KUKA KRL program: MyProgram_197().src

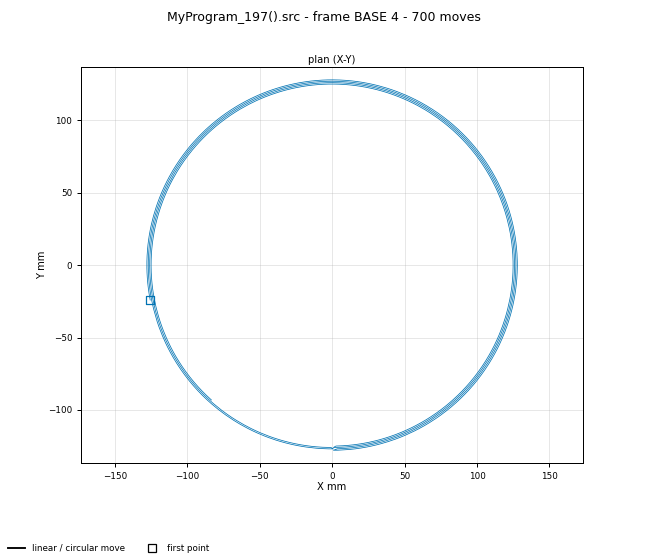
[picture p0: tool path of MyProgram_197().src in frame BASE 4, 700 of 700 moves have a stored position in this frame; points joined in program order, loops and branches not executed]
&ACCESS RVP
&REL 1
&PARAM TEMPLATE = C:\KRC\Roboter\Template\vorgabe
&PARAM EDITMASK = *
DEF MyProgram_197()
; ---- Setting reference (Base) ----
$BASE = BASE_DATA[4]

; --------------------------
; ---- Setting tool (TCP) ----
$TOOL = TOOL_DATA[3]
; --------------------------

$VEL.CP = VEL_APROX_PRINT
Startdeposition()
$VEL.CP = VEL_PRINT
LIN {X -125.5211,Y -24.1311,Z 142,A -173.0115,B 24.959,C -1.4779,E1 24.8425,E2 259.4302} C_DIS
LIN {X -126.2211,Y -20.1609,Z 142,A -174.9442,B 24.959,C -1.4779,E1 24.8416,E2 261.3743} C_DIS
LIN {X -126.7719,Y -16.3344,Z 142,A -176.6253,B 24.9586,C -1.4859,E1 24.841,E2 263.0464} C_DIS
LIN {X -127.2142,Y -12.4288,Z 142,A -178.3522,B 24.9582,C -1.4932,E1 24.8404,E2 264.7662} C_DIS
LIN {X -127.5104,Y -8.8962,Z 142,A 179.9691,B 24.9582,C -1.4943,E1 24.8401,E2 266.4524} C_DIS
LIN {X -127.7137,Y -5.2116,Z 142,A 178.4133,B 24.9576,C -1.5042,E1 24.8399,E2 267.994} C_DIS
LIN {X -127.8085,Y -1.741,Z 142,A 176.7456,B 24.9576,C -1.5042,E1 24.8398,E2 269.6717} C_DIS
LIN {X -127.7955,Y 2.5271,Z 142,A 174.7944,B 24.9573,C -1.5088,E1 24.8398,E2 271.6238} C_DIS
LIN {X -127.6549,Y 6.4899,Z 142,A 173.0449,B 24.9569,C -1.516,E1 24.8401,E2 273.3668} C_DIS
LIN {X -127.3797,Y 10.5984,Z 142,A 171.2555,B 24.9565,C -1.5246,E1 24.8404,E2 275.1463} C_DIS
LIN {X -127.0589,Y 13.9273,Z 142,A 169.9088,B 24.9558,C -1.5365,E1 24.8408,E2 276.4728} C_DIS
LIN {X -126.6556,Y 17.2223,Z 142,A 168.2535,B 24.9559,C -1.5337,E1 24.8414,E2 278.1446} C_DIS
LIN {X -126.1339,Y 20.693,Z 142,A 166.6904,B 24.9556,C -1.5393,E1 24.8421,E2 279.7035} C_DIS
LIN {X -125.5309,Y 24.0797,Z 142,A 165.0614,B 24.9556,C -1.5404,E1 24.8429,E2 281.3395} C_DIS
LIN {X -124.7397,Y 27.8958,Z 142,A 163.305,B 24.9552,C -1.5457,E1 24.8439,E2 283.0938} C_DIS
LIN {X -123.2875,Y 33.7418,Z 142,A 159.7071,B 24.9571,C -1.514,E1 24.8466,E2 286.7881} C_DIS
LIN {X -121.4906,Y 39.7278,Z 142,A 157.6719,B 24.9546,C -1.5574,E1 24.8482,E2 288.7316} C_DIS
LIN {X -120.38,Y 42.9722,Z 142,A 156.2415,B 24.954,C -1.5671,E1 24.8495,E2 290.147} C_DIS
LIN {X -119.1546,Y 46.2598,Z 142,A 154.6827,B 24.9537,C -1.5727,E1 24.8511,E2 291.7012} C_DIS
LIN {X -117.5968,Y 50.0924,Z 142,A 152.5641,B 24.954,C -1.5665,E1 24.8534,E2 293.8465} C_DIS
LIN {X -115.5684,Y 54.6078,Z 142,A 150.536,B 24.9531,C -1.582,E1 24.8557,E2 295.8487} C_DIS
LIN {X -113.9888,Y 57.8302,Z 142,A 148.9277,B 24.9528,C -1.5869,E1 24.8577,E2 297.454} C_DIS
LIN {X -112.4203,Y 60.8282,Z 142,A 147.428,B 24.9525,C -1.5921,E1 24.8597,E2 298.9491} C_DIS
LIN {X -109.9142,Y 65.2469,Z 142,A 145.041,B 24.9525,C -1.5938,E1 24.863,E2 301.3445} C_DIS
LIN {X -107.564,Y 69.0526,Z 142,A 143.0449,B 24.952,C -1.6001,E1 24.866,E2 303.3359} C_DIS
LIN {X -105.1568,Y 72.6668,Z 142,A 141.0404,B 24.9519,C -1.6029,E1 24.8691,E2 305.3436} C_DIS
LIN {X -102.5814,Y 76.2581,Z 142,A 139.0821,B 24.9515,C -1.6095,E1 24.8723,E2 307.2957} C_DIS
LIN {X -99.8212,Y 79.8378,Z 142,A 137.0452,B 24.9512,C -1.6144,E1 24.8758,E2 309.3304} C_DIS
LIN {X -97.6988,Y 82.4216,Z 142,A 135.4913,B 24.9511,C -1.6159,E1 24.8786,E2 310.888} C_DIS
LIN {X -95.3727,Y 85.1019,Z 142,A 133.294,B 24.9525,C -1.5923,E1 24.8829,E2 313.1512} C_DIS
LIN {X -91.7521,Y 88.9933,Z 142,A 130.8212,B 24.9524,C -1.5942,E1 24.8877,E2 315.6302} C_DIS
LIN {X -87.6911,Y 92.9974,Z 142,A 129.1164,B 24.9496,C -1.6394,E1 24.8909,E2 317.2346} C_DIS
LIN {X -85.5377,Y 94.9821,Z 142,A 127.2535,B 24.951,C -1.6171,E1 24.8949,E2 319.1579} C_DIS
LIN {X -82.4213,Y 97.6989,Z 142,A 125.4338,B 24.9507,C -1.6228,E1 24.8987,E2 320.971} C_DIS
LIN {X -79.4084,Y 100.1629,Z 142,A 124.047,B 24.9494,C -1.6432,E1 24.9017,E2 322.3146} C_DIS
LIN {X -76.1096,Y 102.6921,Z 142,A 122.2381,B 24.949,C -1.6497,E1 24.9057,E2 324.1145} C_DIS
LIN {X -73.0168,Y 104.9132,Z 142,A 120.494,B 24.9489,C -1.6515,E1 24.9097,E2 325.8603} C_DIS
LIN {X -69.7238,Y 107.1301,Z 142,A 118.719,B 24.9487,C -1.6552,E1 24.9138,E2 327.6323} C_DIS
LIN {X -66.2948,Y 109.2853,Z 142,A 117.1421,B 24.9477,C -1.6698,E1 24.9175,E2 329.1794} C_DIS
LIN {X -63.6066,Y 110.8718,Z 142,A 115.4076,B 24.9486,C -1.6567,E1 24.9217,E2 330.9504} C_DIS
LIN {X -59.9113,Y 112.9101,Z 142,A 113.5668,B 24.9482,C -1.6624,E1 24.9262,E2 332.7828} C_DIS
LIN {X -56.6117,Y 114.5988,Z 142,A 111.9713,B 24.9478,C -1.6682,E1 24.9302,E2 334.3687} C_DIS
LIN {X -53.8031,Y 115.944,Z 142,A 110.6023,B 24.9476,C -1.6717,E1 24.9336,E2 335.7329} C_DIS
LIN {X -50.9119,Y 117.2424,Z 142,A 109.1599,B 24.9476,C -1.6728,E1 24.9373,E2 337.1761} C_DIS
LIN {X -47.8666,Y 118.5182,Z 142,A 107.9143,B 24.9467,C -1.6861,E1 24.9405,E2 338.393} C_DIS
LIN {X -43.9077,Y 120.0427,Z 142,A 105.6564,B 24.9476,C -1.6717,E1 24.9465,E2 340.6897} C_DIS
LIN {X -40.618,Y 121.1942,Z 142,A 104.4038,B 24.9466,C -1.6884,E1 24.9497,E2 341.9052} C_DIS
LIN {X -36.1428,Y 122.6033,Z 142,A 102.1604,B 24.9468,C -1.6841,E1 24.9557,E2 344.1626} C_DIS
LIN {X -33.0254,Y 123.4793,Z 142,A 100.6082,B 24.9471,C -1.6809,E1 24.9599,E2 345.725} C_DIS
LIN {X -29.441,Y 124.3838,Z 142,A 98.9805,B 24.9469,C -1.6839,E1 24.9643,E2 347.3478} C_DIS
LIN {X -25.4757,Y 125.255,Z 142,A 97.1695,B 24.9467,C -1.6859,E1 24.9692,E2 349.1562} C_DIS
LIN {X -22.4451,Y 125.8335,Z 142,A 95.7361,B 24.9468,C -1.6846,E1 24.9732,E2 350.5942} C_DIS
LIN {X -18.4345,Y 126.4838,Z 142,A 93.8652,B 24.9468,C -1.6835,E1 24.9783,E2 352.4694} C_DIS
LIN {X -14.5682,Y 126.9881,Z 142,A 92.0699,B 24.947,C -1.6822,E1 24.9833,E2 354.2689} C_DIS
LIN {X -10.682,Y 127.3726,Z 142,A 90.406,B 24.9467,C -1.6873,E1 24.9879,E2 355.9217} C_DIS
LIN {X -6.5608,Y 127.6514,Z 142,A 88.2139,B 24.9476,C -1.6716,E1 24.9941,E2 358.1517} C_DIS
LIN {X -3.06,Y 127.7841,Z 142,A 86.8826,B 24.9469,C -1.6835,E1 24.9978,E2 359.4548} C_DIS
LIN {X 0.8422,Y 127.8171,Z 142,A 84.6902,B 24.9482,C -1.6625,E1 25.0041,E2 361.6969} C_DIS
LIN {X 5.3004,Y 127.7102,Z 142,A 83.2635,B 24.9465,C -1.6903,E1 25.0079,E2 363.0573} C_DIS
LIN {X 9.2581,Y 127.484,Z 142,A 81.399,B 24.9467,C -1.686,E1 25.0131,E2 364.9312} C_DIS
LIN {X 13.5575,Y 127.0987,Z 142,A 79.5233,B 24.9466,C -1.6887,E1 25.0183,E2 366.7994} C_DIS
LIN {X 17.3749,Y 126.6352,Z 142,A 77.688,B 24.9469,C -1.6828,E1 25.0234,E2 368.6472} C_DIS
LIN {X 21.1329,Y 126.0605,Z 142,A 76.0592,B 24.9467,C -1.686,E1 25.0278,E2 370.2669} C_DIS
LIN {X 25.2748,Y 125.2959,Z 142,A 74.3916,B 24.9461,C -1.696,E1 25.0323,E2 371.9087} C_DIS
LIN {X 28.2787,Y 124.6522,Z 142,A 72.7974,B 24.9468,C -1.6846,E1 25.0368,E2 373.5279} C_DIS
LIN {X 32.0392,Y 123.7404,Z 142,A 71.1216,B 24.9468,C -1.6864,E1 25.0413,E2 375.1969} C_DIS
LIN {X 35.599,Y 122.7625,Z 142,A 69.4783,B 24.9468,C -1.6859,E1 25.0457,E2 376.8388} C_DIS
LIN {X 38.0718,Y 122.0198,Z 142,A 68.3592,B 24.9467,C -1.6868,E1 25.0487,E2 377.9535} C_DIS
LIN {X 41.211,Y 120.9956,Z 142,A 66.7028,B 24.9473,C -1.6768,E1 25.0531,E2 379.6305} C_DIS
LIN {X 44.792,Y 119.7141,Z 142,A 65.2062,B 24.9468,C -1.6856,E1 25.057,E2 381.1031} C_DIS
LIN {X 50.6604,Y 117.3512,Z 142,A 62.3209,B 24.9471,C -1.6801,E1 25.0645,E2 383.9949} C_DIS
LIN {X 53.5915,Y 116.0419,Z 142,A 60.9427,B 24.9471,C -1.6815,E1 25.0679,E2 385.3665} C_DIS
LIN {X 57.6244,Y 114.0936,Z 142,A 58.835,B 24.9475,C -1.6739,E1 25.0733,E2 387.4864} C_DIS
LIN {X 60.9743,Y 112.3408,Z 142,A 57.0504,B 24.9479,C -1.667,E1 25.0777,E2 389.2823} C_DIS
LIN {X 65.0173,Y 110.0504,Z 142,A 54.8897,B 24.9484,C -1.66,E1 25.0829,E2 391.4529} C_DIS
LIN {X 69.2753,Y 107.4213,Z 142,A 52.7962,B 24.9481,C -1.664,E1 25.0878,E2 393.5303} C_DIS
LIN {X 73.0165,Y 104.9135,Z 142,A 50.8001,B 24.9483,C -1.6618,E1 25.0924,E2 395.5248} C_DIS
LIN {X 76.4508,Y 102.438,Z 142,A 48.8884,B 24.9485,C -1.6577,E1 25.0968,E2 397.4395} C_DIS
LIN {X 79.9444,Y 99.7361,Z 142,A 46.8456,B 24.9489,C -1.6507,E1 25.1013,E2 399.4911} C_DIS
LIN {X 83.3953,Y 96.8683,Z 142,A 44.9121,B 24.9489,C -1.6507,E1 25.1054,E2 401.417} C_DIS
LIN {X 86.719,Y 93.9049,Z 142,A 42.9267,B 24.9492,C -1.6472,E1 25.1095,E2 403.4029} C_DIS
LIN {X 89.7869,Y 90.9764,Z 142,A 40.9805,B 24.9496,C -1.6408,E1 25.1134,E2 405.356} C_DIS
LIN {X 92.8123,Y 87.8873,Z 142,A 39.056,B 24.9498,C -1.6372,E1 25.1171,E2 407.2808} C_DIS
LIN {X 95.8563,Y 84.5567,Z 142,A 37.1194,B 24.9498,C -1.6369,E1 25.1207,E2 409.2094} C_DIS
LIN {X 98.6264,Y 81.309,Z 142,A 35.3653,B 24.9496,C -1.6406,E1 25.1238,E2 410.9469} C_DIS
LIN {X 100.8028,Y 78.595,Z 142,A 33.5657,B 24.9506,C -1.6243,E1 25.127,E2 412.7764} C_DIS
LIN {X 103.5568,Y 74.9283,Z 142,A 31.6066,B 24.9506,C -1.6241,E1 25.1303,E2 414.7265} C_DIS
LIN {X 106.0451,Y 71.3639,Z 142,A 29.6102,B 24.951,C -1.6166,E1 25.1334,E2 416.7309} C_DIS
LIN {X 108.3748,Y 67.7734,Z 142,A 27.867,B 24.9508,C -1.6206,E1 25.136,E2 418.456} C_DIS
LIN {X 110.4975,Y 64.2543,Z 142,A 25.882,B 24.9515,C -1.6081,E1 25.1389,E2 420.46} C_DIS
LIN {X 112.6207,Y 60.4551,Z 142,A 23.9087,B 24.9519,C -1.6015,E1 25.1415,E2 422.4386} C_DIS
LIN {X 114.4624,Y 56.8881,Z 142,A 22.0946,B 24.9523,C -1.5957,E1 25.1438,E2 424.2568} C_DIS
LIN {X 116.4788,Y 52.6375,Z 142,A 20.1062,B 24.9523,C -1.5958,E1 25.1461,E2 426.2341} C_DIS
LIN {X 118.1644,Y 48.7368,Z 142,A 17.8754,B 24.9536,C -1.5732,E1 25.1486,E2 428.506} C_DIS
LIN {X 119.5011,Y 45.3606,Z 142,A 16.5973,B 24.9528,C -1.5865,E1 25.1498,E2 429.7456} C_DIS
LIN {X 120.711,Y 42.032,Z 142,A 15.1443,B 24.9528,C -1.5888,E1 25.1512,E2 431.1852} C_DIS
LIN {X 122.3547,Y 36.9776,Z 142,A 12.5736,B 24.9537,C -1.5716,E1 25.1534,E2 433.7818} C_DIS
LIN {X 123.4571,Y 33.1089,Z 142,A 10.9486,B 24.9535,C -1.5753,E1 25.1546,E2 435.3887} C_DIS
LIN {X 124.253,Y 29.9836,Z 142,A 9.4672,B 24.9539,C -1.5689,E1 25.1556,E2 436.8767} C_DIS
LIN {X 125.0962,Y 26.2549,Z 142,A 7.6746,B 24.9544,C -1.5593,E1 25.1567,E2 438.6815} C_DIS
LIN {X 125.7954,Y 22.6581,Z 142,A 6.1398,B 24.9544,C -1.5597,E1 25.1574,E2 440.2063} C_DIS
LIN {X 126.3274,Y 19.4745,Z 142,A 4.6884,B 24.9547,C -1.5548,E1 25.1581,E2 441.6608} C_DIS
LIN {X 126.8738,Y 15.526,Z 142,A 2.8912,B 24.9551,C -1.5485,E1 25.1587,E2 443.4623} C_DIS
LIN {X 127.2651,Y 11.8982,Z 142,A 1.1815,B 24.9556,C -1.5392,E1 25.1592,E2 445.1836} C_DIS
LIN {X 127.5819,Y 7.7944,Z 142,A -0.2836,B 24.9548,C -1.5533,E1 25.1595,E2 446.607} C_DIS
LIN {X 127.7943,Y 2.5998,Z 142,A -2.9024,B 24.9561,C -1.5303,E1 25.1598,E2 449.2642} C_DIS
LIN {X 127.8184,Y -0.7537,Z 142,A -4.9005,B 24.9579,C -1.4994,E1 25.1598,E2 451.3233} C_DIS
LIN {X 127.7126,Y -5.24,Z 142,A -6.8008,B 24.9579,C -1.4986,E1 25.1595,E2 453.2143} C_DIS
LIN {X 127.4849,Y -9.2456,Z 142,A -8.1262,B 24.9569,C -1.5175,E1 25.1593,E2 454.4872} C_DIS
LIN {X 127.1509,Y -13.0722,Z 142,A -9.9525,B 24.9575,C -1.5063,E1 25.1588,E2 456.3291} C_DIS
LIN {X 126.6224,Y -17.4646,Z 142,A -11.7547,B 24.9573,C -1.5093,E1 25.1582,E2 458.1136} C_DIS
LIN {X 126.2121,Y -20.2188,Z 142,A -13.1455,B 24.958,C -1.4976,E1 25.1576,E2 459.5237} C_DIS
LIN {X 125.5286,Y -24.0917,Z 142,A -14.7731,B 24.958,C -1.499,E1 25.1568,E2 461.1385} C_DIS
LIN {X 124.7218,Y -27.9739,Z 142,A -16.5708,B 24.9583,C -1.4921,E1 25.1557,E2 462.9419} C_DIS
LIN {X 123.9309,Y -31.2888,Z 142,A -18.0523,B 24.9584,C -1.4896,E1 25.1547,E2 464.4208} C_DIS
LIN {X 123.1029,Y -34.402,Z 142,A -19.499,B 24.9587,C -1.4848,E1 25.1537,E2 465.8705} C_DIS
LIN {X 121.7562,Y -38.9003,Z 142,A -21.5091,B 24.9587,C -1.483,E1 25.152,E2 467.8734} C_DIS
LIN {X 120.8724,Y -41.5664,Z 142,A -22.6636,B 24.9587,C -1.4845,E1 25.151,E2 469.0179} C_DIS
LIN {X 119.2673,Y -45.9699,Z 142,A -25.5916,B 24.9615,C -1.4344,E1 25.148,E2 472.0476} C_DIS
LIN {X 117.3926,Y -50.5645,Z 142,A -27.6944,B 24.9615,C -1.4338,E1 25.1457,E2 474.1403} C_DIS
LIN {X 115.5438,Y -54.6593,Z 142,A -29.2089,B 24.9604,C -1.4538,E1 25.144,E2 475.5996} C_DIS
LIN {X 113.976,Y -57.8555,Z 142,A -30.7502,B 24.9605,C -1.4518,E1 25.1421,E2 477.1373} C_DIS
LIN {X 112.2793,Y -61.0871,Z 142,A -32.4087,B 24.9608,C -1.4456,E1 25.1399,E2 478.8016} C_DIS
LIN {X 110.2445,Y -64.6869,Z 142,A -34.2573,B 24.9611,C -1.4404,E1 25.1373,E2 480.6529} C_DIS
LIN {X 107.9456,Y -68.4548,Z 142,A -36.8227,B 24.9631,C -1.404,E1 25.1334,E2 483.2912} C_DIS
LIN {X 105.1875,Y -72.6221,Z 142,A -38.4797,B 24.9618,C -1.428,E1 25.1309,E2 484.8835} C_DIS
LIN {X 102.7157,Y -76.0778,Z 142,A -40.3737,B 24.9621,C -1.4232,E1 25.1278,E2 486.7796} C_DIS
LIN {X 99.8994,Y -79.7395,Z 142,A -42.7564,B 24.9632,C -1.4013,E1 25.1236,E2 489.2029} C_DIS
LIN {X 97.5112,Y -82.6429,Z 142,A -44.2335,B 24.9629,C -1.4076,E1 25.121,E2 490.6583} C_DIS
LIN {X 94.3141,Y -86.2739,Z 142,A -46.2515,B 24.9628,C -1.4098,E1 25.1172,E2 492.6621} C_DIS
LIN {X 91.4762,Y -89.2773,Z 142,A -48.1018,B 24.963,C -1.4052,E1 25.1136,E2 494.5152} C_DIS
LIN {X 88.7083,Y -92.028,Z 142,A -49.9167,B 24.9634,C -1.3975,E1 25.11,E2 496.3409} C_DIS
LIN {X 85.397,Y -95.1085,Z 142,A -51.8738,B 24.9634,C -1.3963,E1 25.106,E2 498.2929} C_DIS
LIN {X 82.0889,Y -97.9779,Z 142,A -53.7796,B 24.9636,C -1.3947,E1 25.1019,E2 500.1949} C_DIS
LIN {X 79.0225,Y -100.4674,Z 142,A -55.7429,B 24.9643,C -1.3808,E1 25.0976,E2 502.1838} C_DIS
LIN {X 74.8412,Y -103.6199,Z 142,A -57.9197,B 24.9641,C -1.3845,E1 25.0927,E2 504.3439} C_DIS
LIN {X 71.4919,Y -105.9584,Z 142,A -59.5222,B 24.9637,C -1.3926,E1 25.0891,E2 505.9219} C_DIS
LIN {X 67.4024,Y -108.6056,Z 142,A -61.9092,B 24.9644,C -1.3778,E1 25.0834,E2 508.3361} C_DIS
LIN {X 63.7647,Y -110.7809,Z 142,A -63.7764,B 24.9645,C -1.3759,E1 25.0789,E2 510.2021} C_DIS
LIN {X 60.2915,Y -112.7086,Z 142,A -65.5892,B 24.9648,C -1.3711,E1 25.0745,E2 512.021} C_DIS
LIN {X 56.7055,Y -114.5525,Z 142,A -67.2969,B 24.9647,C -1.3732,E1 25.0702,E2 513.7192} C_DIS
LIN {X 53.6446,Y -116.0173,Z 142,A -68.7914,B 24.9647,C -1.3721,E1 25.0665,E2 515.2124} C_DIS
LIN {X 50.9167,Y -117.2404,Z 142,A -70.604,B 24.9661,C -1.3459,E1 25.0617,E2 517.0824} C_DIS
LIN {X 47.1355,Y -118.8129,Z 142,A -72.1159,B 24.9654,C -1.3597,E1 25.0579,E2 518.5583} C_DIS
LIN {X 43.615,Y -120.1482,Z 142,A -73.5663,B 24.9649,C -1.3695,E1 25.0541,E2 519.9824} C_DIS
LIN {X 38.4751,Y -121.892,Z 142,A -76.206,B 24.9656,C -1.3559,E1 25.0471,E2 522.6493} C_DIS
LIN {X 33.9823,Y -123.2202,Z 142,A -78.2965,B 24.9656,C -1.354,E1 25.0415,E2 524.7407} C_DIS
LIN {X 30.1126,Y -124.2219,Z 142,A -79.9655,B 24.9654,C -1.3584,E1 25.037,E2 526.3969} C_DIS
LIN {X 27.1122,Y -124.9111,Z 142,A -81.3455,B 24.9655,C -1.3571,E1 25.0332,E2 527.7781} C_DIS
LIN {X 23.7699,Y -125.5902,Z 142,A -82.9365,B 24.9657,C -1.3526,E1 25.0288,E2 529.3778} C_DIS
LIN {X 19.7669,Y -126.2821,Z 142,A -84.7048,B 24.9657,C -1.3539,E1 25.024,E2 531.1413} C_DIS
LIN {X 16.1602,Y -126.7948,Z 142,A -86.226,B 24.9654,C -1.3584,E1 25.0198,E2 532.6505} C_DIS
LIN {X 11.938,Y -127.2613,Z 142,A -88.2251,B 24.9657,C -1.3525,E1 25.0142,E2 534.6622} C_DIS
LIN {X 4.0063,Y -127.7578,Z 142,A -91.6254,B 24.9654,C -1.3591,E1 25.0048,E2 538.0457} C_DIS
LIN {X 0.9092,Y -127.7876,Z 142,A -93.0254,B 24.9654,C -1.3586,E1 25.0009,E2 539.4466} C_DIS
Enddeposition()
LIN {X 0.9092,Y -127.7876,Z 142,A -93.0254,B 24.9654,C -1.3586,E1 25.0009,E2 539.4466} C_DIS
Startdeposition()
$VEL.CP = VEL_PRINT
LIN {X 3.5824,Y -126.8,Z 142,A -91.1897,B 24.4984,C -1.3089,E1 24.537,E2 537.666} C_DIS
LIN {X 9.8682,Y -126.4677,Z 142,A -88.1818,B 24.498,C -1.3182,E1 24.5455,E2 534.6369} C_DIS
LIN {X 12.9375,Y -126.1906,Z 142,A -86.8649,B 24.4981,C -1.3153,E1 24.5491,E2 533.328} C_DIS
LIN {X 16.3259,Y -125.7956,Z 142,A -85.3641,B 24.4981,C -1.3143,E1 24.5533,E2 531.8307} C_DIS
LIN {X 20.2934,Y -125.218,Z 142,A -83.4855,B 24.4979,C -1.3189,E1 24.5585,E2 529.9428} C_DIS
LIN {X 23.9684,Y -124.5655,Z 142,A -81.8724,B 24.498,C -1.3167,E1 24.5629,E2 528.3369} C_DIS
LIN {X 28.0075,Y -123.72,Z 142,A -80.0259,B 24.498,C -1.3176,E1 24.5679,E2 526.4907} C_DIS
LIN {X 31.241,Y -122.9431,Z 142,A -78.5522,B 24.498,C -1.3176,E1 24.5719,E2 525.0191} C_DIS
LIN {X 34.1426,Y -122.169,Z 142,A -76.8134,B 24.4969,C -1.3383,E1 24.5767,E2 523.2335} C_DIS
LIN {X 37.5906,Y -121.1535,Z 142,A -75.6621,B 24.4981,C -1.3165,E1 24.5797,E2 522.1368} C_DIS
LIN {X 44.5342,Y -118.7757,Z 142,A -72.2474,B 24.4976,C -1.3257,E1 24.5887,E2 518.7069} C_DIS
LIN {X 47.4707,Y -117.6329,Z 142,A -70.2624,B 24.496,C -1.3562,E1 24.594,E2 516.6532} C_DIS
LIN {X 51.6656,Y -115.8517,Z 142,A -68.7876,B 24.4974,C -1.3297,E1 24.5976,E2 515.2457} C_DIS
LIN {X 54.574,Y -114.5104,Z 142,A -67.3594,B 24.4974,C -1.3311,E1 24.6012,E2 513.818} C_DIS
LIN {X 57.4301,Y -113.105,Z 142,A -65.9894,B 24.4974,C -1.3301,E1 24.6046,E2 512.4541} C_DIS
LIN {X 60.4982,Y -111.4965,Z 142,A -64.2484,B 24.4968,C -1.3417,E1 24.609,E2 510.6903} C_DIS
LIN {X 64.3963,Y -109.2912,Z 142,A -62.2671,B 24.4967,C -1.3433,E1 24.6137,E2 508.7112} C_DIS
LIN {X 68.0897,Y -107.0296,Z 142,A -60.3105,B 24.4965,C -1.3471,E1 24.6184,E2 506.7519} C_DIS
LIN {X 75.4232,Y -101.9947,Z 142,A -55.6797,B 24.4944,C -1.3869,E1 24.6291,E2 502.0419} C_DIS
LIN {X 79.5373,Y -98.8192,Z 142,A -53.9974,B 24.4959,C -1.3578,E1 24.6326,E2 500.4359} C_DIS
LIN {X 82.7212,Y -96.1698,Z 142,A -52.1009,B 24.4956,C -1.3634,E1 24.6367,E2 498.5335} C_DIS
LIN {X 86.0309,Y -93.221,Z 142,A -49.7721,B 24.4945,C -1.385,E1 24.6416,E2 496.1624} C_DIS
LIN {X 88.7862,Y -90.6004,Z 142,A -48.3236,B 24.495,C -1.3753,E1 24.6444,E2 494.7434} C_DIS
LIN {X 92.0815,Y -87.2496,Z 142,A -46.2633,B 24.495,C -1.3774,E1 24.6484,E2 492.687} C_DIS
LIN {X 94.7896,Y -84.3,Z 142,A -44.0129,B 24.4934,C -1.405,E1 24.6527,E2 490.3807} C_DIS
LIN {X 97.7119,Y -80.8938,Z 142,A -41.8235,B 24.4927,C -1.4189,E1 24.6566,E2 488.1683} C_DIS
LIN {X 101.0638,Y -76.6654,Z 142,A -40.0221,B 24.4941,C -1.3925,E1 24.6596,E2 486.439} C_DIS
LIN {X 103.4919,Y -73.3547,Z 142,A -37.2766,B 24.4913,C -1.4442,E1 24.6642,E2 483.5831} C_DIS
LIN {X 107.259,Y -67.7268,Z 142,A -35.1816,B 24.4936,C -1.4025,E1 24.6672,E2 481.5988} C_DIS
LIN {X 109.5043,Y -64.0336,Z 142,A -33.2445,B 24.4933,C -1.4075,E1 24.6699,E2 479.66} C_DIS
LIN {X 111.5832,Y -60.3384,Z 142,A -31.2807,B 24.4929,C -1.4157,E1 24.6726,E2 477.6869} C_DIS
LIN {X 113.6319,Y -56.3809,Z 142,A -29.4244,B 24.4929,C -1.4137,E1 24.6749,E2 475.8456} C_DIS
LIN {X 116.1307,Y -51.0383,Z 142,A -26.3133,B 24.4912,C -1.4452,E1 24.6786,E2 472.6762} C_DIS
LIN {X 117.6366,Y -47.4613,Z 142,A -25.0374,B 24.4923,C -1.4257,E1 24.6799,E2 471.454} C_DIS
LIN {X 118.7903,Y -44.4951,Z 142,A -23.4782,B 24.4917,C -1.4366,E1 24.6814,E2 469.8778} C_DIS
LIN {X 120.3455,Y -40.0991,Z 142,A -21.558,B 24.4919,C -1.4336,E1 24.6832,E2 467.9757} C_DIS
LIN {X 121.8318,Y -35.3286,Z 142,A -19.1706,B 24.4911,C -1.4476,E1 24.6851,E2 465.5687} C_DIS
LIN {X 122.9124,Y -31.3619,Z 142,A -17.3901,B 24.491,C -1.4496,E1 24.6864,E2 463.7939} C_DIS
LIN {X 124.3904,Y -24.864,Z 142,A -14.3701,B 24.4904,C -1.4598,E1 24.6882,E2 460.7672} C_DIS
LIN {X 125.1064,Y -20.9624,Z 142,A -12.6537,B 24.4904,C -1.4618,E1 24.689,E2 459.0564} C_DIS
LIN {X 125.6936,Y -17.1039,Z 142,A -10.8449,B 24.4899,C -1.4699,E1 24.6897,E2 457.239} C_DIS
LIN {X 126.1566,Y -13.2533,Z 142,A -9.1161,B 24.4896,C -1.4745,E1 24.6903,E2 455.5096} C_DIS
LIN {X 126.5133,Y -9.2427,Z 142,A -7.3882,B 24.4896,C -1.4757,E1 24.6907,E2 453.7892} C_DIS
LIN {X 126.6899,Y -6.3824,Z 142,A -6.0741,B 24.4892,C -1.481,E1 24.6909,E2 452.4704} C_DIS
LIN {X 126.8523,Y -0.221,Z 142,A -3.1948,B 24.4884,C -1.4951,E1 24.691,E2 449.575} C_DIS
LIN {X 126.8205,Y 2.8402,Z 142,A -1.7619,B 24.488,C -1.5022,E1 24.691,E2 448.1337} C_DIS
LIN {X 126.6321,Y 7.4489,Z 142,A 0.1586,B 24.4881,C -1.5005,E1 24.6907,E2 446.2288} C_DIS
LIN {X 126.3715,Y 11.0191,Z 142,A 1.7934,B 24.4878,C -1.5067,E1 24.6903,E2 444.5891} C_DIS
LIN {X 125.9469,Y 15.1138,Z 142,A 3.6221,B 24.4875,C -1.5112,E1 24.6897,E2 442.7608} C_DIS
LIN {X 125.4053,Y 19.0953,Z 142,A 5.4185,B 24.4872,C -1.516,E1 24.689,E2 440.9636} C_DIS
LIN {X 124.8109,Y 22.6572,Z 142,A 7.0659,B 24.4869,C -1.5221,E1 24.6882,E2 439.3115} C_DIS
LIN {X 124.0247,Y 26.625,Z 142,A 8.838,B 24.4867,C -1.525,E1 24.6872,E2 437.5429} C_DIS
LIN {X 123.2119,Y 30.1668,Z 142,A 10.5459,B 24.4862,C -1.5336,E1 24.6861,E2 435.8245} C_DIS
LIN {X 122.0531,Y 34.557,Z 142,A 12.7063,B 24.4855,C -1.5457,E1 24.6845,E2 433.6479} C_DIS
LIN {X 119.6097,Y 42.2497,Z 142,A 16.1784,B 24.4854,C -1.5477,E1 24.6815,E2 430.1909} C_DIS
LIN {X 118.4151,Y 45.4869,Z 142,A 18.0658,B 24.4841,C -1.5694,E1 24.6796,E2 428.2622} C_DIS
LIN {X 117.0646,Y 48.8552,Z 142,A 19.2367,B 24.4852,C -1.5501,E1 24.6784,E2 427.1443} C_DIS
LIN {X 115.8591,Y 51.6491,Z 142,A 20.6227,B 24.4849,C -1.5547,E1 24.6768,E2 425.7549} C_DIS
LIN {X 114.5182,Y 54.5577,Z 142,A 21.8499,B 24.4854,C -1.5476,E1 24.6754,E2 424.5515} C_DIS
LIN {X 112.3862,Y 58.8243,Z 142,A 24.2286,B 24.4843,C -1.5651,E1 24.6724,E2 422.1436} C_DIS
LIN {X 110.4489,Y 62.3902,Z 142,A 26.6547,B 24.4822,C -1.6007,E1 24.669,E2 419.645} C_DIS
LIN {X 108.0931,Y 66.3875,Z 142,A 28.2209,B 24.4835,C -1.5791,E1 24.6668,E2 418.1389} C_DIS
LIN {X 105.8225,Y 69.9505,Z 142,A 30.1266,B 24.4832,C -1.584,E1 24.6639,E2 416.2312} C_DIS
LIN {X 103.0731,Y 73.9417,Z 142,A 32.2953,B 24.4829,C -1.5886,E1 24.6604,E2 414.0623} C_DIS
LIN {X 100.5596,Y 77.3259,Z 142,A 34.6128,B 24.4813,C -1.6144,E1 24.6564,E2 411.694} C_DIS
LIN {X 97.9495,Y 80.6068,Z 142,A 36.1038,B 24.4823,C -1.5984,E1 24.6538,E2 410.2485} C_DIS
LIN {X 95.1553,Y 83.8863,Z 142,A 38.0355,B 24.4821,C -1.6022,E1 24.6503,E2 408.3165} C_DIS
LIN {X 92.0474,Y 87.2857,Z 142,A 40.1122,B 24.4818,C -1.6068,E1 24.6463,E2 406.2383} C_DIS
LIN {X 89.0172,Y 90.3738,Z 142,A 42.0526,B 24.4816,C -1.6103,E1 24.6425,E2 404.2977} C_DIS
LIN {X 85.8642,Y 93.3743,Z 142,A 43.9871,B 24.4814,C -1.6128,E1 24.6386,E2 402.3652} C_DIS
LIN {X 82.5232,Y 96.3403,Z 142,A 46.0216,B 24.4811,C -1.6177,E1 24.6343,E2 400.3272} C_DIS
LIN {X 79.2929,Y 99.0162,Z 142,A 48.0599,B 24.4804,C -1.6286,E1 24.6298,E2 398.2707} C_DIS
LIN {X 75.2785,Y 102.101,Z 142,A 50.1812,B 24.4807,C -1.6244,E1 24.6251,E2 396.1673} C_DIS
LIN {X 69.7179,Y 105.9756,Z 142,A 53.2073,B 24.4805,C -1.6278,E1 24.6182,E2 393.1436} C_DIS
LIN {X 66.044,Y 108.3038,Z 142,A 54.9102,B 24.4811,C -1.6178,E1 24.6142,E2 391.4701} C_DIS
LIN {X 62.3499,Y 110.4715,Z 142,A 57.123,B 24.4801,C -1.6345,E1 24.6088,E2 389.2241} C_DIS
LIN {X 58.2891,Y 112.6672,Z 142,A 59.534,B 24.4789,C -1.6535,E1 24.6027,E2 386.7742} C_DIS
LIN {X 54.9449,Y 114.3332,Z 142,A 60.7932,B 24.4801,C -1.6344,E1 24.5997,E2 385.5644} C_DIS
LIN {X 51.8867,Y 115.7529,Z 142,A 62.2838,B 24.4801,C -1.6346,E1 24.5959,E2 384.0771} C_DIS
LIN {X 48.8191,Y 117.0797,Z 142,A 63.7163,B 24.4801,C -1.6325,E1 24.5922,E2 382.6532} C_DIS
LIN {X 43.6792,Y 119.0943,Z 142,A 66.3995,B 24.4795,C -1.6442,E1 24.5852,E2 379.9478} C_DIS
LIN {X 37.6714,Y 121.1286,Z 142,A 69.2528,B 24.4793,C -1.646,E1 24.5776,E2 377.0956} C_DIS
LIN {X 33.9626,Y 122.2193,Z 142,A 70.919,B 24.4795,C -1.6434,E1 24.5731,E2 375.4387} C_DIS
LIN {X 30.0308,Y 123.2447,Z 142,A 72.7369,B 24.4795,C -1.6436,E1 24.5682,E2 373.6228} C_DIS
LIN {X 25.9731,Y 124.1648,Z 142,A 74.7166,B 24.4791,C -1.6495,E1 24.5628,E2 371.6318} C_DIS
LIN {X 22.3487,Y 124.8661,Z 142,A 76.2706,B 24.4794,C -1.6447,E1 24.5586,E2 370.0911} C_DIS
LIN {X 18.5986,Y 125.4813,Z 142,A 78.0519,B 24.4792,C -1.6483,E1 24.5536,E2 368.3028} C_DIS
LIN {X 15.0671,Y 125.9525,Z 142,A 79.6192,B 24.4793,C -1.6467,E1 24.5493,E2 366.7407} C_DIS
LIN {X 10.9197,Y 126.3799,Z 142,A 81.446,B 24.4795,C -1.6442,E1 24.5442,E2 364.9211} C_DIS
LIN {X 7.2461,Y 126.6446,Z 142,A 83.1931,B 24.4792,C -1.6482,E1 24.5394,E2 363.1651} C_DIS
LIN {X 4.3731,Y 126.7765,Z 142,A 84.3862,B 24.4795,C -1.643,E1 24.5361,E2 361.9847} C_DIS
LIN {X 0.0789,Y 126.8521,Z 142,A 86.4757,B 24.4791,C -1.6499,E1 24.5302,E2 359.8789} C_DIS
LIN {X -3.7927,Y 126.7942,Z 142,A 88.2504,B 24.4791,C -1.6507,E1 24.5252,E2 358.1022} C_DIS
LIN {X -8.2647,Y 126.5819,Z 142,A 90.2832,B 24.4791,C -1.6504,E1 24.5196,E2 356.0694} C_DIS
LIN {X -12.2289,Y 126.2597,Z 142,A 91.9669,B 24.4795,C -1.6442,E1 24.5149,E2 354.3998} C_DIS
LIN {X -16.2897,Y 125.8003,Z 142,A 93.8163,B 24.4795,C -1.6433,E1 24.5098,E2 352.5513} C_DIS
LIN {X -19.9453,Y 125.2737,Z 142,A 95.5872,B 24.4793,C -1.647,E1 24.5049,E2 350.77} C_DIS
LIN {X -23.5766,Y 124.6403,Z 142,A 97.1514,B 24.4797,C -1.6409,E1 24.5006,E2 349.2187} C_DIS
LIN {X -26.6103,Y 124.0279,Z 142,A 98.6655,B 24.4794,C -1.6452,E1 24.4964,E2 347.6924} C_DIS
LIN {X -31.2164,Y 122.9493,Z 142,A 100.6823,B 24.4799,C -1.6375,E1 24.491,E2 345.6913} C_DIS
LIN {X -34.9253,Y 121.9498,Z 142,A 102.3815,B 24.4801,C -1.634,E1 24.4864,E2 343.9979} C_DIS
LIN {X -40.1923,Y 120.3144,Z 142,A 104.9348,B 24.4801,C -1.634,E1 24.4796,E2 341.4401} C_DIS
LIN {X -43.399,Y 119.1958,Z 142,A 106.7868,B 24.4793,C -1.6468,E1 24.4747,E2 339.5531} C_DIS
LIN {X -46.5764,Y 117.9917,Z 142,A 108.0529,B 24.4802,C -1.6322,E1 24.4715,E2 338.3198} C_DIS
LIN {X -49.8897,Y 116.6285,Z 142,A 109.5845,B 24.4806,C -1.6258,E1 24.4676,E2 336.7998} C_DIS
LIN {X -53.561,Y 114.9882,Z 142,A 111.4998,B 24.4805,C -1.6276,E1 24.4627,E2 334.8754} C_DIS
LIN {X -57.2282,Y 113.2078,Z 142,A 113.266,B 24.4809,C -1.6212,E1 24.4583,E2 333.1201} C_DIS
LIN {X -60.4658,Y 111.5142,Z 142,A 114.9248,B 24.4811,C -1.6187,E1 24.4542,E2 331.4625} C_DIS
LIN {X -66.0409,Y 108.3057,Z 142,A 117.9958,B 24.4809,C -1.621,E1 24.4468,E2 328.3765} C_DIS
LIN {X -69.9502,Y 105.8227,Z 142,A 120.0608,B 24.4812,C -1.6158,E1 24.4419,E2 326.3174} C_DIS
LIN {X -73.3665,Y 103.4837,Z 142,A 121.8876,B 24.4816,C -1.61,E1 24.4378,E2 324.4983} C_DIS
LIN {X -76.58,Y 101.1284,Z 142,A 123.7337,B 24.4816,C -1.6083,E1 24.4336,E2 322.6494} C_DIS
LIN {X -79.9401,Y 98.4944,Z 142,A 125.5622,B 24.4822,C -1.5995,E1 24.4297,E2 320.8353} C_DIS
LIN {X -82.3113,Y 96.5209,Z 142,A 127.5209,B 24.4808,C -1.6223,E1 24.4254,E2 318.8138} C_DIS
LIN {X -85.5626,Y 93.6514,Z 142,A 129.0799,B 24.4822,C -1.5993,E1 24.4222,E2 317.3039} C_DIS
LIN {X -88.552,Y 90.8301,Z 142,A 131.3388,B 24.4814,C -1.6132,E1 24.4176,E2 315.0017} C_DIS
LIN {X -91.5167,Y 87.8418,Z 142,A 133.2332,B 24.4817,C -1.6082,E1 24.414,E2 313.1111} C_DIS
LIN {X -94.3325,Y 84.8106,Z 142,A 134.7107,B 24.4831,C -1.5856,E1 24.4113,E2 311.6818} C_DIS
LIN {X -96.6886,Y 82.1142,Z 142,A 136.3272,B 24.4833,C -1.5813,E1 24.4084,E2 310.068} C_DIS
LIN {X -99.5126,Y 78.669,Z 142,A 138.4015,B 24.4835,C -1.5788,E1 24.4047,E2 307.99} C_DIS
LIN {X -102.1995,Y 75.1444,Z 142,A 140.3566,B 24.484,C -1.5712,E1 24.4015,E2 306.0437} C_DIS
LIN {X -104.7864,Y 71.4936,Z 142,A 142.413,B 24.4842,C -1.5671,E1 24.3982,E2 303.9869} C_DIS
LIN {X -107.1337,Y 67.9254,Z 142,A 144.3604,B 24.4845,C -1.5624,E1 24.3952,E2 302.0407} C_DIS
LIN {X -109.4672,Y 64.0966,Z 142,A 147.2318,B 24.4825,C -1.5949,E1 24.3911,E2 299.0753} C_DIS
LIN {X -112.4928,Y 58.6213,Z 142,A 149.2608,B 24.4852,C -1.5504,E1 24.3885,E2 297.1434} C_DIS
LIN {X -114.5354,Y 54.5216,Z 142,A 151.9547,B 24.4839,C -1.5724,E1 24.3852,E2 294.3812} C_DIS
LIN {X -116.7597,Y 49.5853,Z 142,A 153.8019,B 24.486,C -1.5377,E1 24.3832,E2 292.6077} C_DIS
LIN {X -118.1879,Y 46.0716,Z 142,A 155.4015,B 24.4866,C -1.5273,E1 24.3816,E2 291.0241} C_DIS
LIN {X -119.3361,Y 43.0099,Z 142,A 156.8587,B 24.4869,C -1.5218,E1 24.3802,E2 289.5719} C_DIS
LIN {X -120.5646,Y 39.441,Z 142,A 158.8266,B 24.4865,C -1.5282,E1 24.3784,E2 287.5771} C_DIS
LIN {X -122.1743,Y 34.1238,Z 142,A 161.1386,B 24.4875,C -1.5113,E1 24.3766,E2 285.2923} C_DIS
LIN {X -123.07,Y 30.7408,Z 142,A 162.9052,B 24.4873,C -1.5146,E1 24.3754,E2 283.5073} C_DIS
LIN {X -124.1911,Y 25.8438,Z 142,A 165.096,B 24.4879,C -1.5037,E1 24.3741,E2 281.3297} C_DIS
LIN {X -124.8858,Y 22.2387,Z 142,A 166.6727,B 24.4885,C -1.4947,E1 24.3733,E2 279.7653} C_DIS
LIN {X -125.5278,Y 18.273,Z 142,A 169.0863,B 24.4872,C -1.5157,E1 24.3723,E2 277.2861} C_DIS
LIN {X -126.0981,Y 13.7976,Z 142,A 170.5687,B 24.4891,C -1.484,E1 24.3719,E2 275.8715} C_DIS
LIN {X -126.4359,Y 10.2564,Z 142,A 172.2742,B 24.4891,C -1.4832,E1 24.3714,E2 274.1576} C_DIS
LIN {X -126.6953,Y 6.2739,Z 142,A 174.0154,B 24.4896,C -1.4745,E1 24.3711,E2 272.4266} C_DIS
LIN {X -126.8276,Y 2.4378,Z 142,A 175.7403,B 24.4899,C -1.4684,E1 24.3711,E2 270.7059} C_DIS
LIN {X -126.8474,Y -1.0413,Z 142,A 177.4585,B 24.4899,C -1.4699,E1 24.3711,E2 268.9736} C_DIS
LIN {X -126.7549,Y -4.9266,Z 142,A 179.1167,B 24.4904,C -1.4598,E1 24.3711,E2 267.3296} C_DIS
LIN {X -126.5357,Y -8.9368,Z 142,A -179.0594,B 24.4907,C -1.4543,E1 24.3715,E2 265.5077} C_DIS
LIN {X -126.242,Y -12.413,Z 142,A -177.3773,B 24.4907,C -1.454,E1 24.3719,E2 263.8162} C_DIS
LIN {X -125.7733,Y -16.4955,Z 142,A -175.6212,B 24.4913,C -1.4435,E1 24.3725,E2 262.0747} C_DIS
LIN {X -125.1917,Y -20.451,Z 142,A -173.6128,B 24.4912,C -1.4469,E1 24.3734,E2 260.046} C_DIS
LIN {X -124.529,Y -24.159,Z 142,A -171.2022,B 24.4897,C -1.4737,E1 24.3748,E2 257.5558} C_DIS
LIN {X -123.2319,Y -30.0838,Z 142,A -169.4683,B 24.4927,C -1.4194,E1 24.3758,E2 255.9431} C_DIS
LIN {X -120.703,Y -39.0123,Z 142,A -165.0282,B 24.4927,C -1.4176,E1 24.3793,E2 251.4813} C_DIS
LIN {X -119.3993,Y -42.8347,Z 142,A -163.2968,B 24.4933,C -1.4079,E1 24.3808,E2 249.7634} C_DIS
LIN {X -118.2609,Y -45.8839,Z 142,A -161.8154,B 24.4935,C -1.404,E1 24.3823,E2 248.2829} C_DIS
LIN {X -117.1336,Y -48.69,Z 142,A -160.4593,B 24.4937,C -1.3995,E1 24.3837,E2 246.9299} C_DIS
LIN {X -116.0928,Y -51.1267,Z 142,A -159.1116,B 24.4936,C -1.4028,E1 24.3853,E2 245.5666} C_DIS
LIN {X -114.9534,Y -53.6363,Z 142,A -157.6252,B 24.4932,C -1.4103,E1 24.3871,E2 244.0539} C_DIS
LIN {X -113.4953,Y -56.6561,Z 142,A -156.3629,B 24.494,C -1.3945,E1 24.3886,E2 242.8229} C_DIS
LIN {X -111.7865,Y -59.96,Z 142,A -154.6454,B 24.4942,C -1.3915,E1 24.3908,E2 241.1033} C_DIS
LIN {X -109.6084,Y -63.8555,Z 142,A -152.6052,B 24.4944,C -1.3871,E1 24.3936,E2 239.0629} C_DIS
LIN {X -107.3642,Y -67.5602,Z 142,A -150.8724,B 24.4952,C -1.3716,E1 24.3961,E2 237.3585} C_DIS
LIN {X -104.4798,Y -71.9403,Z 142,A -148.1874,B 24.4948,C -1.3799,E1 24.4004,E2 234.6397} C_DIS
LIN {X -101.6474,Y -75.8898,Z 142,A -145.904,B 24.4948,C -1.3785,E1 24.4042,E2 232.3486} C_DIS
LIN {X -98.4438,Y -80.0022,Z 142,A -143.6659,B 24.4954,C -1.3674,E1 24.408,E2 230.1266} C_DIS
LIN {X -95.4816,Y -83.5147,Z 142,A -141.6345,B 24.4958,C -1.3605,E1 24.4117,E2 228.1025} C_DIS
LIN {X -92.5696,Y -86.732,Z 142,A -139.6286,B 24.4959,C -1.3582,E1 24.4155,E2 226.0932} C_DIS
LIN {X -89.5918,Y -89.8042,Z 142,A -137.682,B 24.4961,C -1.3546,E1 24.4193,E2 224.1466} C_DIS
LIN {X -86.3323,Y -92.9418,Z 142,A -135.664,B 24.4964,C -1.3492,E1 24.4234,E2 222.1333} C_DIS
LIN {X -83.1279,Y -95.8191,Z 142,A -133.8892,B 24.497,C -1.3374,E1 24.4271,E2 220.38} C_DIS
LIN {X -78.4536,Y -99.6818,Z 142,A -131.0418,B 24.497,C -1.3372,E1 24.4333,E2 217.522} C_DIS
LIN {X -73.4861,Y -103.3989,Z 142,A -128.1504,B 24.497,C -1.3364,E1 24.4398,E2 214.6221} C_DIS
LIN {X -70.1362,Y -105.6998,Z 142,A -126.3154,B 24.4972,C -1.3333,E1 24.444,E2 212.7883} C_DIS
LIN {X -67.8431,Y -107.1856,Z 142,A -124.4893,B 24.4959,C -1.3594,E1 24.4485,E2 210.8932} C_DIS
LIN {X -63.6126,Y -109.7491,Z 142,A -122.821,B 24.4974,C -1.3293,E1 24.4524,E2 209.2926} C_DIS
LIN {X -58.0342,Y -112.7974,Z 142,A -119.9657,B 24.4976,C -1.3246,E1 24.4594,E2 206.4403} C_DIS
LIN {X -54.6606,Y -114.469,Z 142,A -118.3677,B 24.498,C -1.3177,E1 24.4634,E2 204.8549} C_DIS
LIN {X -51.755,Y -115.8118,Z 142,A -117.0537,B 24.4984,C -1.3098,E1 24.4667,E2 203.5566} C_DIS
LIN {X -46.8834,Y -117.8688,Z 142,A -114.3702,B 24.4978,C -1.3213,E1 24.4737,E2 200.8392} C_DIS
LIN {X -43.9994,Y -118.976,Z 142,A -113.1293,B 24.4982,C -1.3126,E1 24.4769,E2 199.6167} C_DIS
LIN {X -39.0134,Y -120.7026,Z 142,A -110.6515,B 24.4982,C -1.3151,E1 24.4834,E2 197.1281} C_DIS
LIN {X -35.6675,Y -121.7325,Z 142,A -109.099,B 24.4982,C -1.3126,E1 24.4876,E2 195.5789} C_DIS
LIN {X -31.9754,Y -122.7563,Z 142,A -107.2541,B 24.498,C -1.317,E1 24.4926,E2 193.7206} C_DIS
LIN {X -28.312,Y -123.6504,Z 142,A -105.6993,B 24.4984,C -1.3089,E1 24.4968,E2 192.1831} C_DIS
LIN {X -24.8492,Y -124.3935,Z 142,A -103.9474,B 24.4981,C -1.3156,E1 24.5016,E2 190.413} C_DIS
LIN {X -20.9952,Y -125.1009,Z 142,A -102.3284,B 24.4985,C -1.3077,E1 24.506,E2 188.8115} C_DIS
LIN {X -17.7348,Y -125.6047,Z 142,A -100.706,B 24.4982,C -1.3137,E1 24.5105,E2 187.1731} C_DIS
LIN {X -13.5014,Y -126.1299,Z 142,A -98.9515,B 24.4986,C -1.3051,E1 24.5154,E2 185.4383} C_DIS
LIN {X -10.7758,Y -126.392,Z 142,A -97.5037,B 24.4981,C -1.3153,E1 24.5195,E2 183.9652} C_DIS
LIN {X -7.5867,Y -126.6236,Z 142,A -95.5283,B 24.4968,C -1.3414,E1 24.5252,E2 181.9261} C_DIS
LIN {X -2.5433,Y -126.8259,Z 142,A -93.8736,B 24.4983,C -1.3109,E1 24.5296,E2 180.3448} C_DIS
LIN {X 0.8963,Y -126.8363,Z 142,A -92.3785,B 24.4984,C -1.3086,E1 24.5337,E2 178.8553} C_DIS
Enddeposition()
LIN {X 0.8963,Y -126.8363,Z 142,A -92.3785,B 24.4984,C -1.3086,E1 24.5337,E2 178.8553} C_DIS
Startdeposition()
$VEL.CP = VEL_PRINT
LIN {X -0.8273,Y -125.8788,Z 142,A -93.715,B 23.845,C -1.1662,E1 23.8699,E2 180.4512} C_DIS
LIN {X -6.5882,Y -125.7091,Z 142,A -96.2437,B 23.8448,C -1.1704,E1 23.8628,E2 182.9701} C_DIS
LIN {X -10.9105,Y -125.408,Z 142,A -98.1624,B 23.8448,C -1.1729,E1 23.8575,E2 184.8834} C_DIS
LIN {X -13.967,Y -125.105,Z 142,A -99.7716,B 23.8451,C -1.1633,E1 23.853,E2 186.5174} C_DIS
LIN {X -17.8518,Y -124.609,Z 142,A -101.4436,B 23.8449,C -1.1688,E1 23.8484,E2 188.1772} C_DIS
LIN {X -21.4858,Y -124.0359,Z 142,A -103.2201,B 23.8451,C -1.1646,E1 23.8435,E2 189.9658} C_DIS
LIN {X -25.1472,Y -123.3437,Z 142,A -104.7986,B 23.8448,C -1.1707,E1 23.8392,E2 191.531} C_DIS
LIN {X -28.9423,Y -122.5101,Z 142,A -106.6545,B 23.8449,C -1.1676,E1 23.8341,E2 193.3972} C_DIS
LIN {X -32.5088,Y -121.6109,Z 142,A -108.2438,B 23.8447,C -1.1725,E1 23.8298,E2 194.9768} C_DIS
LIN {X -36.2405,Y -120.5531,Z 142,A -110.1857,B 23.845,C -1.1656,E1 23.8246,E2 196.9389} C_DIS
LIN {X -40.7096,Y -119.1178,Z 142,A -112.0384,B 23.8444,C -1.1803,E1 23.8197,E2 198.759} C_DIS
LIN {X -43.75,Y -118.0344,Z 142,A -113.6751,B 23.8446,C -1.174,E1 23.8154,E2 200.4148} C_DIS
LIN {X -49.4626,Y -115.7572,Z 142,A -116.3093,B 23.8442,C -1.1843,E1 23.8086,E2 203.0296} C_DIS
LIN {X -52.9317,Y -114.2114,Z 142,A -118.1585,B 23.8443,C -1.1808,E1 23.8039,E2 204.8921} C_DIS
LIN {X -55.9257,Y -112.7757,Z 142,A -119.6695,B 23.8443,C -1.1827,E1 23.8001,E2 206.4026} C_DIS
LIN {X -60.8771,Y -110.1837,Z 142,A -122.2004,B 23.8441,C -1.1866,E1 23.7939,E2 208.9312} C_DIS
LIN {X -66.4824,Y -106.8951,Z 142,A -125.0415,B 23.8436,C -1.1961,E1 23.7871,E2 211.7577} C_DIS
LIN {X -69.0144,Y -105.2784,Z 142,A -126.6509,B 23.844,C -1.1875,E1 23.7832,E2 213.3941} C_DIS
LIN {X -72.4558,Y -102.94,Z 142,A -129.0636,B 23.8449,C -1.1678,E1 23.7776,E2 215.8644} C_DIS
LIN {X -76.157,Y -100.2334,Z 142,A -130.6948,B 23.8438,C -1.1915,E1 23.774,E2 217.4427} C_DIS
LIN {X -81.9802,Y -95.5288,Z 142,A -134.0922,B 23.8435,C -1.1984,E1 23.7667,E2 220.8366} C_DIS
LIN {X -85.289,Y -92.5865,Z 142,A -136.1021,B 23.8433,C -1.2027,E1 23.7626,E2 222.8443} C_DIS
LIN {X -88.4359,Y -89.5863,Z 142,A -138.1187,B 23.8432,C -1.2052,E1 23.7585,E2 224.8635} C_DIS
LIN {X -91.3934,Y -86.5665,Z 142,A -140.0267,B 23.8429,C -1.2102,E1 23.7548,E2 226.768} C_DIS
LIN {X -94.1727,Y -83.5345,Z 142,A -141.9319,B 23.8429,C -1.213,E1 23.7513,E2 228.6752} C_DIS
LIN {X -97.1702,Y -80.0282,Z 142,A -143.9861,B 23.8425,C -1.2199,E1 23.7476,E2 230.7222} C_DIS
LIN {X -100.3236,Y -76.0375,Z 142,A -146.1519,B 23.8419,C -1.232,E1 23.7439,E2 232.8686} C_DIS
LIN {X -102.2549,Y -73.4197,Z 142,A -147.8077,B 23.8421,C -1.2281,E1 23.7411,E2 234.5426} C_DIS
LIN {X -105.8148,Y -68.1897,Z 142,A -150.4537,B 23.8412,C -1.2456,E1 23.7371,E2 237.1589} C_DIS
LIN {X -108.1792,Y -64.3719,Z 142,A -152.7922,B 23.8416,C -1.2383,E1 23.7336,E2 239.5282} C_DIS
LIN {X -110.3637,Y -60.5508,Z 142,A -154.63,B 23.841,C -1.2509,E1 23.7311,E2 241.3448} C_DIS
LIN {X -111.8808,Y -57.6984,Z 142,A -156.5529,B 23.8417,C -1.2356,E1 23.7286,E2 243.3167} C_DIS
LIN {X -113.3742,Y -54.7034,Z 142,A -157.833,B 23.841,C -1.2503,E1 23.727,E2 244.5674} C_DIS
LIN {X -114.9076,Y -51.4027,Z 142,A -159.3544,B 23.8405,C -1.2609,E1 23.7253,E2 246.0713} C_DIS
LIN {X -116.1684,Y -48.486,Z 142,A -160.8351,B 23.8403,C -1.2636,E1 23.7237,E2 247.5538} C_DIS
LIN {X -117.3595,Y -45.5275,Z 142,A -162.3039,B 23.8402,C -1.2671,E1 23.7222,E2 249.0226} C_DIS
LIN {X -118.6171,Y -42.1467,Z 142,A -164.0438,B 23.8402,C -1.2678,E1 23.7205,E2 250.7712} C_DIS
LIN {X -119.8537,Y -38.4858,Z 142,A -166.7629,B 23.8419,C -1.2325,E1 23.7181,E2 253.5944} C_DIS
LIN {X -121.7294,Y -32.0647,Z 142,A -168.8091,B 23.8393,C -1.284,E1 23.7167,E2 255.5249} C_DIS
LIN {X -122.8918,Y -27.2721,Z 142,A -171.4526,B 23.8398,C -1.2741,E1 23.715,E2 258.2095} C_DIS
LIN {X -123.6142,Y -23.7826,Z 142,A -172.8,B 23.839,C -1.2908,E1 23.7143,E2 259.5237} C_DIS
LIN {X -124.253,Y -20.1879,Z 142,A -174.313,B 23.8384,C -1.3024,E1 23.7136,E2 261.0173} C_DIS
LIN {X -124.7677,Y -16.7099,Z 142,A -176.031,B 23.8384,C -1.3025,E1 23.7129,E2 262.7459} C_DIS
LIN {X -125.2369,Y -12.7397,Z 142,A -177.9442,B 23.8383,C -1.3043,E1 23.7123,E2 264.6666} C_DIS
LIN {X -125.5691,Y -8.865,Z 142,A -179.7032,B 23.8379,C -1.3105,E1 23.7119,E2 266.4214} C_DIS
LIN {X -125.7908,Y -4.7756,Z 142,A 178.4814,B 23.8375,C -1.3186,E1 23.7117,E2 268.2281} C_DIS
LIN {X -125.881,Y -0.5685,Z 142,A 176.6285,B 23.8371,C -1.3275,E1 23.7117,E2 270.0707} C_DIS
LIN {X -125.8396,Y 3.2543,Z 142,A 174.8232,B 23.8369,C -1.3304,E1 23.7117,E2 271.8803} C_DIS
LIN {X -125.6846,Y 7.0679,Z 142,A 172.9787,B 23.8369,C -1.3315,E1 23.712,E2 273.7338} C_DIS
LIN {X -125.4162,Y 10.8137,Z 142,A 171.3613,B 23.8364,C -1.3409,E1 23.7123,E2 275.3379} C_DIS
LIN {X -124.987,Y 14.9785,Z 142,A 168.8905,B 23.8373,C -1.3233,E1 23.7131,E2 277.868} C_DIS
LIN {X -124.3855,Y 19.3475,Z 142,A 167.4772,B 23.8356,C -1.3548,E1 23.7137,E2 279.2118} C_DIS
LIN {X -123.8577,Y 22.4816,Z 142,A 165.9222,B 23.8356,C -1.3549,E1 23.7144,E2 280.7763} C_DIS
LIN {X -122.8948,Y 27.2659,Z 142,A 163.6165,B 23.8354,C -1.3585,E1 23.7158,E2 283.0875} C_DIS
LIN {X -122.0155,Y 30.9557,Z 142,A 161.9986,B 23.8349,C -1.3686,E1 23.7168,E2 284.6901} C_DIS
LIN {X -121.1579,Y 34.1594,Z 142,A 160.4889,B 23.8346,C -1.3734,E1 23.7179,E2 286.1972} C_DIS
LIN {X -119.6056,Y 39.2533,Z 142,A 158.0969,B 23.8341,C -1.3824,E1 23.7199,E2 288.5813} C_DIS
LIN {X -118.3903,Y 42.7755,Z 142,A 156.3598,B 23.8339,C -1.386,E1 23.7215,E2 290.3198} C_DIS
LIN {X -117.2133,Y 45.9036,Z 142,A 154.8163,B 23.8337,C -1.3897,E1 23.7231,E2 291.8631} C_DIS
LIN {X -115.7508,Y 49.4774,Z 142,A 152.1183,B 23.8356,C -1.3555,E1 23.7262,E2 294.662} C_DIS
LIN {X -113.2067,Y 55.052,Z 142,A 150.1829,B 23.8332,C -1.3998,E1 23.7284,E2 296.4982} C_DIS
LIN {X -108.7977,Y 63.3215,Z 142,A 145.8257,B 23.8327,C -1.4084,E1 23.7342,E2 300.8583} C_DIS
LIN {X -106.6159,Y 66.9299,Z 142,A 143.8657,B 23.8325,C -1.4122,E1 23.737,E2 302.8196} C_DIS
LIN {X -104.0587,Y 70.8404,Z 142,A 141.7328,B 23.8322,C -1.4179,E1 23.7403,E2 304.9494} C_DIS
LIN {X -101.5493,Y 74.3924,Z 142,A 139.7611,B 23.8318,C -1.4237,E1 23.7435,E2 306.9169} C_DIS
LIN {X -98.8733,Y 77.9138,Z 142,A 137.723,B 23.8316,C -1.428,E1 23.747,E2 308.9545} C_DIS
LIN {X -96.1796,Y 81.2162,Z 142,A 135.7656,B 23.8313,C -1.4323,E1 23.7505,E2 310.9107} C_DIS
LIN {X -93.3982,Y 84.3997,Z 142,A 133.6534,B 23.8315,C -1.4292,E1 23.7545,E2 313.0406} C_DIS
LIN {X -88.9988,Y 89.0271,Z 142,A 130.9011,B 23.8307,C -1.4429,E1 23.7598,E2 315.7712} C_DIS
LIN {X -85.8357,Y 92.0798,Z 142,A 128.9325,B 23.8304,C -1.4491,E1 23.7637,E2 317.7331} C_DIS
LIN {X -80.5823,Y 96.7114,Z 142,A 125.7707,B 23.8299,C -1.4574,E1 23.7704,E2 320.8873} C_DIS
LIN {X -77.4088,Y 99.2697,Z 142,A 123.8195,B 23.8299,C -1.4573,E1 23.7747,E2 322.8464} C_DIS
LIN {X -74.0358,Y 101.8096,Z 142,A 121.9602,B 23.8295,C -1.464,E1 23.7788,E2 324.6959} C_DIS
LIN {X -70.8117,Y 104.0781,Z 142,A 120.0929,B 23.8295,C -1.4644,E1 23.7831,E2 326.5689} C_DIS
LIN {X -66.9609,Y 106.5963,Z 142,A 117.9934,B 23.8293,C -1.4682,E1 23.7881,E2 328.6661} C_DIS
LIN {X -63.7831,Y 108.5273,Z 142,A 115.8632,B 23.8302,C -1.4522,E1 23.7933,E2 330.8427} C_DIS
LIN {X -59.9715,Y 110.6798,Z 142,A 114.3314,B 23.8289,C -1.4757,E1 23.7969,E2 332.3209} C_DIS
LIN {X -56.9637,Y 112.2548,Z 142,A 112.8785,B 23.8285,C -1.4823,E1 23.8005,E2 333.7614} C_DIS
LIN {X -53.4034,Y 113.9933,Z 142,A 111.1376,B 23.8281,C -1.4879,E1 23.8048,E2 335.4933} C_DIS
LIN {X -49.7289,Y 115.6421,Z 142,A 109.1959,B 23.8283,C -1.4858,E1 23.8098,E2 337.445} C_DIS
LIN {X -46.1609,Y 117.1133,Z 142,A 107.0994,B 23.829,C -1.4733,E1 23.8154,E2 339.5775} C_DIS
LIN {X -43.0518,Y 118.2907,Z 142,A 105.9751,B 23.8279,C -1.4924,E1 23.8182,E2 340.6567} C_DIS
LIN {X -36.0147,Y 120.621,Z 142,A 102.6182,B 23.8276,C -1.4971,E1 23.8271,E2 344.0085} C_DIS
LIN {X -33.9673,Y 121.2116,Z 142,A 101.2812,B 23.8285,C -1.4818,E1 23.8308,E2 345.3855} C_DIS
LIN {X -27.2785,Y 122.8921,Z 142,A 98.4754,B 23.8275,C -1.4996,E1 23.8383,E2 348.1514} C_DIS
LIN {X -24.2862,Y 123.5179,Z 142,A 96.9284,B 23.8278,C -1.4938,E1 23.8426,E2 349.7145} C_DIS
LIN {X -20.5547,Y 124.1918,Z 142,A 95.2733,B 23.8275,C -1.4982,E1 23.8471,E2 351.3603} C_DIS
LIN {X -16.3588,Y 124.8137,Z 142,A 93.3514,B 23.8275,C -1.4999,E1 23.8524,E2 353.2798} C_DIS
LIN {X -12.2482,Y 125.2842,Z 142,A 91.4644,B 23.8274,C -1.5007,E1 23.8576,E2 355.166} C_DIS
LIN {X -8.2596,Y 125.6111,Z 142,A 89.4541,B 23.8278,C -1.4929,E1 23.8633,E2 357.1963} C_DIS
LIN {X -3.5892,Y 125.8302,Z 142,A 87.4897,B 23.8274,C -1.501,E1 23.8687,E2 359.1411} C_DIS
LIN {X 0.6657,Y 125.8797,Z 142,A 85.3253,B 23.828,C -1.4911,E1 23.8748,E2 361.3301} C_DIS
LIN {X 5.0973,Y 125.7783,Z 142,A 83.5005,B 23.8274,C -1.5,E1 23.8799,E2 363.1323} C_DIS
LIN {X 9.2377,Y 125.5419,Z 142,A 81.6724,B 23.8273,C -1.5026,E1 23.8849,E2 364.953} C_DIS
LIN {X 13.1958,Y 125.188,Z 142,A 79.8621,B 23.8273,C -1.5023,E1 23.89,E2 366.763} C_DIS
LIN {X 16.7088,Y 124.7679,Z 142,A 78.2909,B 23.8273,C -1.5038,E1 23.8943,E2 368.3292} C_DIS
LIN {X 20.5504,Y 124.1925,Z 142,A 76.491,B 23.8273,C -1.5018,E1 23.8993,E2 370.1324} C_DIS
LIN {X 23.8765,Y 123.5963,Z 142,A 74.9224,B 23.8274,C -1.4997,E1 23.9036,E2 371.7041} C_DIS
LIN {X 28.4333,Y 122.6286,Z 142,A 72.9317,B 23.8272,C -1.5046,E1 23.909,E2 373.6799} C_DIS
LIN {X 31.0867,Y 121.9823,Z 142,A 71.5819,B 23.8275,C -1.4989,E1 23.9127,E2 375.0417} C_DIS
LIN {X 35.3433,Y 120.8176,Z 142,A 69.7368,B 23.8271,C -1.5051,E1 23.9176,E2 376.8683} C_DIS
LIN {X 37.7157,Y 120.0997,Z 142,A 68.564,B 23.8273,C -1.5021,E1 23.9207,E2 378.0463} C_DIS
LIN {X 41.1161,Y 118.9769,Z 142,A 66.8823,B 23.8275,C -1.4983,E1 23.9252,E2 379.7338} C_DIS
LIN {X 47.2114,Y 116.6924,Z 142,A 63.891,B 23.8278,C -1.4941,E1 23.933,E2 382.7289} C_DIS
LIN {X 50.1477,Y 115.461,Z 142,A 62.484,B 23.8278,C -1.4944,E1 23.9366,E2 384.1315} C_DIS
LIN {X 52.9949,Y 114.1821,Z 142,A 61.0377,B 23.8279,C -1.4916,E1 23.9403,E2 385.581} C_DIS
LIN {X 58.5536,Y 111.4337,Z 142,A 58.3605,B 23.8277,C -1.4948,E1 23.947,E2 388.2427} C_DIS
LIN {X 63.7181,Y 108.5655,Z 142,A 55.6066,B 23.8281,C -1.4878,E1 23.9537,E2 391.0052} C_DIS
LIN {X 66.8049,Y 106.6944,Z 142,A 53.7919,B 23.8288,C -1.4771,E1 23.958,E2 392.8403} C_DIS
LIN {X 71.554,Y 103.5684,Z 142,A 51.0568,B 23.8294,C -1.4659,E1 23.9644,E2 395.5934} C_DIS
LIN {X 74.7432,Y 101.2916,Z 142,A 49.4137,B 23.8292,C -1.4694,E1 23.9681,E2 397.2217} C_DIS
LIN {X 78.139,Y 98.6958,Z 142,A 47.4993,B 23.8293,C -1.4672,E1 23.9723,E2 399.1339} C_DIS
LIN {X 81.4668,Y 95.9668,Z 142,A 45.5652,B 23.8295,C -1.4646,E1 23.9765,E2 401.0666} C_DIS
LIN {X 84.7842,Y 93.0492,Z 142,A 43.5614,B 23.8297,C -1.4609,E1 23.9806,E2 403.0712} C_DIS
LIN {X 87.8978,Y 90.1141,Z 142,A 41.6148,B 23.8299,C -1.4568,E1 23.9846,E2 405.0193} C_DIS
LIN {X 90.8788,Y 87.1065,Z 142,A 39.6918,B 23.8302,C -1.4528,E1 23.9883,E2 406.9435} C_DIS
LIN {X 93.9404,Y 83.7957,Z 142,A 37.6723,B 23.8304,C -1.4497,E1 23.9921,E2 408.9612} C_DIS
LIN {X 96.7281,Y 80.5622,Z 142,A 35.4734,B 23.8313,C -1.4328,E1 23.9961,E2 411.1911} C_DIS
LIN {X 98.8392,Y 77.9567,Z 142,A 34.1801,B 23.8309,C -1.4404,E1 23.9983,E2 412.4595} C_DIS
LIN {X 100.7765,Y 75.4364,Z 142,A 32.727,B 23.8311,C -1.4365,E1 24.0008,E2 413.9148} C_DIS
LIN {X 103.2463,Y 72.0186,Z 142,A 31.1199,B 23.8305,C -1.4468,E1 24.0033,E2 415.4883} C_DIS
LIN {X 104.9192,Y 69.56,Z 142,A 29.4807,B 23.8315,C -1.4294,E1 24.0059,E2 417.1619} C_DIS
LIN {X 107.2964,Y 65.8328,Z 142,A 26.6349,B 23.8341,C -1.3838,E1 24.0102,E2 420.1047} C_DIS
LIN {X 110.5443,Y 60.2198,Z 142,A 23.9314,B 23.8338,C -1.3876,E1 24.0138,E2 422.784} C_DIS
LIN {X 112.9636,Y 55.5448,Z 142,A 22.3277,B 23.8321,C -1.4193,E1 24.0157,E2 424.3005} C_DIS
LIN {X 114.3158,Y 52.7059,Z 142,A 20.915,B 23.8323,C -1.4161,E1 24.0174,E2 425.713} C_DIS
LIN {X 115.5707,Y 49.8941,Z 142,A 19.4997,B 23.8325,C -1.4114,E1 24.019,E2 427.1318} C_DIS
LIN {X 117.4363,Y 45.33,Z 142,A 17.2976,B 23.8328,C -1.4068,E1 24.0213,E2 429.3323} C_DIS
LIN {X 118.4949,Y 42.4857,Z 142,A 15.8751,B 23.8331,C -1.4007,E1 24.0226,E2 430.7616} C_DIS
LIN {X 119.7473,Y 38.8167,Z 142,A 14.159,B 23.8333,C -1.3977,E1 24.0242,E2 432.4747} C_DIS
LIN {X 121.3654,Y 33.4176,Z 142,A 11.6073,B 23.8337,C -1.3905,E1 24.0262,E2 435.0288} C_DIS
LIN {X 122.3045,Y 29.7951,Z 142,A 9.8402,B 23.8341,C -1.3821,E1 24.0274,E2 436.8059} C_DIS
LIN {X 123.1175,Y 26.2343,Z 142,A 8.2721,B 23.8341,C -1.3816,E1 24.0283,E2 438.3658} C_DIS
LIN {X 123.8556,Y 22.4938,Z 142,A 6.4854,B 23.8346,C -1.3735,E1 24.0293,E2 440.1611} C_DIS
LIN {X 124.4101,Y 19.1887,Z 142,A 5.0087,B 23.8347,C -1.3711,E1 24.0299,E2 441.6347} C_DIS
LIN {X 124.9417,Y 15.3577,Z 142,A 3.1783,B 23.8352,C -1.362,E1 24.0306,E2 443.4761} C_DIS
LIN {X 125.373,Y 11.3233,Z 142,A 1.28,B 23.8357,C -1.3535,E1 24.0311,E2 445.3835} C_DIS
LIN {X 125.6828,Y 7.0965,Z 142,A -0.8208,B 23.8365,C -1.3388,E1 24.0315,E2 447.5074} C_DIS
LIN {X 125.8573,Y 2.4987,Z 142,A -2.6274,B 23.8361,C -1.3462,E1 24.0316,E2 449.2844} C_DIS
LIN {X 125.8729,Y -1.557,Z 142,A -5.0696,B 23.8379,C -1.3108,E1 24.0316,E2 451.7983} C_DIS
LIN {X 125.7177,Y -6.4177,Z 142,A -6.4694,B 23.8362,C -1.3437,E1 24.0314,E2 453.1083} C_DIS
LIN {X 125.5435,Y -9.2163,Z 142,A -7.8958,B 23.8368,C -1.3321,E1 24.0311,E2 454.5544} C_DIS
LIN {X 125.1867,Y -13.2076,Z 142,A -9.7179,B 23.8371,C -1.3263,E1 24.0306,E2 456.3795} C_DIS
LIN {X 124.7499,Y -16.8456,Z 142,A -11.3346,B 23.8373,C -1.3233,E1 24.0301,E2 457.9934} C_DIS
LIN {X 124.2299,Y -20.3264,Z 142,A -12.9833,B 23.8377,C -1.3158,E1 24.0294,E2 459.6504} C_DIS
LIN {X 123.6104,Y -23.8026,Z 142,A -14.7227,B 23.8383,C -1.3041,E1 24.0285,E2 461.4079} C_DIS
LIN {X 122.1755,Y -30.3253,Z 142,A -17.4757,B 23.8381,C -1.3085,E1 24.0268,E2 464.1332} C_DIS
LIN {X 121.2093,Y -33.9755,Z 142,A -19.8391,B 23.84,C -1.2712,E1 24.025,E2 466.5741} C_DIS
LIN {X 119.8995,Y -38.3422,Z 142,A -20.9827,B 23.8379,C -1.3107,E1 24.0241,E2 467.6138} C_DIS
LIN {X 118.2658,Y -43.1209,Z 142,A -23.5688,B 23.8391,C -1.2891,E1 24.0217,E2 470.2376} C_DIS
LIN {X 117.1899,Y -45.9638,Z 142,A -24.9423,B 23.8392,C -1.2853,E1 24.0203,E2 471.6125} C_DIS
LIN {X 116.0823,Y -48.6922,Z 142,A -26.3393,B 23.8396,C -1.2783,E1 24.0188,E2 473.0185} C_DIS
LIN {X 113.6333,Y -54.1615,Z 142,A -28.7181,B 23.8391,C -1.2873,E1 24.0161,E2 475.3615} C_DIS
LIN {X 111.8657,Y -57.728,Z 142,A -30.9445,B 23.8405,C -1.2613,E1 24.0133,E2 477.6395} C_DIS
LIN {X 109.7292,Y -61.6925,Z 142,A -32.9169,B 23.8405,C -1.259,E1 24.0106,E2 479.6066} C_DIS
LIN {X 107.5376,Y -65.4389,Z 142,A -34.8642,B 23.8408,C -1.2547,E1 24.0078,E2 481.5541} C_DIS
LIN {X 103.3101,Y -71.927,Z 142,A -38.3364,B 23.8411,C -1.2472,E1 24.0025,E2 485.0263} C_DIS
LIN {X 100.9777,Y -75.1663,Z 142,A -40.7778,B 23.8429,C -1.2117,E1 23.9983,E2 487.5429} C_DIS
LIN {X 97.9649,Y -79.0527,Z 142,A -42.1938,B 23.8412,C -1.2459,E1 23.996,E2 488.8676} C_DIS
LIN {X 94.653,Y -82.9899,Z 142,A -44.7509,B 23.842,C -1.2291,E1 23.9913,E2 491.4538} C_DIS
LIN {X 89.314,Y -88.71,Z 142,A -47.9914,B 23.8417,C -1.2359,E1 23.9852,E2 494.6628} C_DIS
LIN {X 84.7184,Y -93.109,Z 142,A -50.829,B 23.8419,C -1.2317,E1 23.9795,E2 497.4983} C_DIS
LIN {X 81.6985,Y -95.7698,Z 142,A -52.9907,B 23.8429,C -1.2113,E1 23.9748,E2 499.7012} C_DIS
LIN {X 79.669,Y -97.4644,Z 142,A -54.3556,B 23.8434,C -1.2008,E1 23.9718,E2 501.0867} C_DIS
LIN {X 75.9176,Y -100.4141,Z 142,A -56.38,B 23.8433,C -1.2033,E1 23.9674,E2 503.0971} C_DIS
LIN {X 69.1624,Y -105.1809,Z 142,A -60.054,B 23.8434,C -1.1999,E1 23.959,E2 506.7662} C_DIS
LIN {X 65.7051,Y -107.3747,Z 142,A -61.9542,B 23.8437,C -1.1946,E1 23.9545,E2 508.6731} C_DIS
LIN {X 62.0288,Y -109.5401,Z 142,A -63.9502,B 23.844,C -1.1884,E1 23.9496,E2 510.6779} C_DIS
LIN {X 58.4879,Y -111.4682,Z 142,A -65.6663,B 23.8439,C -1.191,E1 23.9454,E2 512.3825} C_DIS
LIN {X 55.5855,Y -112.9436,Z 142,A -67.1074,B 23.8439,C -1.1905,E1 23.9418,E2 513.8207} C_DIS
LIN {X 52.7605,Y -114.2905,Z 142,A -68.5951,B 23.8441,C -1.1852,E1 23.938,E2 515.3174} C_DIS
LIN {X 48.2731,Y -116.2574,Z 142,A -70.7404,B 23.8441,C -1.186,E1 23.9326,E2 517.4555} C_DIS
LIN {X 44.9008,Y -117.6031,Z 142,A -72.9489,B 23.8454,C -1.1572,E1 23.9266,E2 519.7299} C_DIS
LIN {X 40.9345,Y -119.0398,Z 142,A -74.4974,B 23.8447,C -1.1724,E1 23.9226,E2 521.2377} C_DIS
LIN {X 35.8276,Y -120.6754,Z 142,A -76.9333,B 23.8448,C -1.1697,E1 23.9161,E2 523.6755} C_DIS
LIN {X 31.2421,Y -121.9428,Z 142,A -78.9376,B 23.8446,C -1.1751,E1 23.9108,E2 525.6632} C_DIS
LIN {X 28.0776,Y -122.7098,Z 142,A -80.3819,B 23.8446,C -1.1754,E1 23.9069,E2 527.1044} C_DIS
LIN {X 24.6745,Y -123.4399,Z 142,A -82.0095,B 23.8447,C -1.172,E1 23.9024,E2 528.7385} C_DIS
LIN {X 20.8055,Y -124.1499,Z 142,A -83.7525,B 23.8447,C -1.1728,E1 23.8976,E2 530.4774} C_DIS
LIN {X 17.3039,Y -124.6873,Z 142,A -85.5955,B 23.8453,C -1.1609,E1 23.8924,E2 532.3481} C_DIS
LIN {X 13.4217,Y -125.1637,Z 142,A -87.142,B 23.8448,C -1.1708,E1 23.8882,E2 533.869} C_DIS
LIN {X 9.6184,Y -125.5141,Z 142,A -89.2602,B 23.8457,C -1.1522,E1 23.8822,E2 536.032} C_DIS
LIN {X 6.1871,Y -125.7293,Z 142,A -90.7228,B 23.8455,C -1.1563,E1 23.8782,E2 537.4838} C_DIS
LIN {X 0.8953,Y -125.877,Z 142,A -92.8313,B 23.8448,C -1.1697,E1 23.8724,E2 539.559} C_DIS
Enddeposition()
LIN {X 0.8953,Y -125.877,Z 142,A -92.8313,B 23.8448,C -1.1697,E1 23.8724,E2 539.559} C_DIS
Startdeposition()
$VEL.CP = VEL_PRINT
LIN {X 2.6952,Y -124.8846,Z 142,A -91.0232,B 23.1289,C -1.0932,E1 23.1586,E2 537.8485} C_DIS
LIN {X 7.2544,Y -124.702,Z 142,A -88.9532,B 23.1289,C -1.093,E1 23.1644,E2 535.7799} C_DIS
LIN {X 11.1351,Y -124.4163,Z 142,A -87.2262,B 23.129,C -1.0912,E1 23.1692,E2 534.0585} C_DIS
LIN {X 14.6513,Y -124.0499,Z 142,A -85.6389,B 23.129,C -1.0906,E1 23.1736,E2 532.474} C_DIS
LIN {X 18.5818,Y -123.5233,Z 142,A -83.7674,B 23.1289,C -1.0942,E1 23.1788,E2 530.5951} C_DIS
LIN {X 22.0313,Y -122.9537,Z 142,A -82.2133,B 23.1289,C -1.0931,E1 23.183,E2 529.0455} C_DIS
LIN {X 25.7111,Y -122.239,Z 142,A -80.4494,B 23.1288,C -1.0966,E1 23.1879,E2 527.275} C_DIS
LIN {X 29.2488,Y -121.4392,Z 142,A -78.8611,B 23.1288,C -1.0948,E1 23.1922,E2 525.6939} C_DIS
LIN {X 32.7431,Y -120.5454,Z 142,A -76.6205,B 23.1276,C -1.1237,E1 23.1984,E2 523.3836} C_DIS
LIN {X 37.1019,Y -119.2759,Z 142,A -75.04,B 23.1285,C -1.1027,E1 23.2025,E2 521.8595} C_DIS
LIN {X 39.7935,Y -118.4042,Z 142,A -73.2814,B 23.1275,C -1.1258,E1 23.2073,E2 520.0459} C_DIS
LIN {X 43.9012,Y -116.9429,Z 142,A -71.7948,B 23.1284,C -1.1045,E1 23.211,E2 518.617} C_DIS
LIN {X 47.8074,Y -115.4015,Z 142,A -69.9575,B 23.1284,C -1.103,E1 23.2157,E2 516.788} C_DIS
LIN {X 50.9493,Y -114.0487,Z 142,A -68.1665,B 23.1279,C -1.1158,E1 23.2204,E2 514.9694} C_DIS
LIN {X 55.0582,Y -112.123,Z 142,A -66.2778,B 23.1282,C -1.11,E1 23.2251,E2 513.1007} C_DIS
LIN {X 58.0783,Y -110.5885,Z 142,A -64.8438,B 23.1283,C -1.107,E1 23.2286,E2 511.6786} C_DIS
LIN {X 61.4418,Y -108.7583,Z 142,A -62.914,B 23.1278,C -1.1182,E1 23.2334,E2 509.7266} C_DIS
LIN {X 64.783,Y -106.8016,Z 142,A -61.1983,B 23.1278,C -1.1186,E1 23.2375,E2 508.0155} C_DIS
LIN {X 68.2723,Y -104.6058,Z 142,A -59.2631,B 23.1275,C -1.1244,E1 23.2421,E2 506.0727} C_DIS
LIN {X 72.3655,Y -101.8171,Z 142,A -56.9998,B 23.1273,C -1.1285,E1 23.2473,E2 503.8073} C_DIS
LIN {X 75.592,Y -99.4454,Z 142,A -55.1319,B 23.1271,C -1.1339,E1 23.2515,E2 501.9332} C_DIS
LIN {X 78.9423,Y -96.8066,Z 142,A -53.4673,B 23.1275,C -1.1243,E1 23.255,E2 500.2996} C_DIS
LIN {X 81.1001,Y -95.0064,Z 142,A -51.6688,B 23.1263,C -1.1515,E1 23.259,E2 498.4399} C_DIS
LIN {X 83.6595,Y -92.761,Z 142,A -50.3386,B 23.1266,C -1.144,E1 23.2617,E2 497.1343} C_DIS
LIN {X 86.868,Y -89.7627,Z 142,A -48.4656,B 23.1267,C -1.1421,E1 23.2655,E2 495.2747} C_DIS
LIN {X 89.7222,Y -86.9097,Z 142,A -46.1609,B 23.1255,C -1.1684,E1 23.2701,E2 492.9141} C_DIS
LIN {X 92.4112,Y -84.0451,Z 142,A -44.7506,B 23.1261,C -1.1541,E1 23.2726,E2 491.5468} C_DIS
LIN {X 95.1995,Y -80.873,Z 142,A -42.9255,B 23.1261,C -1.1537,E1 23.276,E2 489.7316} C_DIS
LIN {X 98.2938,Y -77.0826,Z 142,A -40.4169,B 23.1253,C -1.1724,E1 23.2804,E2 487.1886} C_DIS
LIN {X 101.3307,Y -73.045,Z 142,A -38.2768,B 23.1253,C -1.1701,E1 23.2839,E2 485.0654} C_DIS
LIN {X 103.6406,Y -69.729,Z 142,A -36.6677,B 23.1257,C -1.1635,E1 23.2864,E2 483.4815} C_DIS
LIN {X 106.0029,Y -66.0816,Z 142,A -34.4518,B 23.1249,C -1.1799,E1 23.2898,E2 481.2364} C_DIS
LIN {X 108.3105,Y -62.2284,Z 142,A -32.4147,B 23.1247,C -1.1847,E1 23.2927,E2 479.1985} C_DIS
LIN {X 110.2278,Y -58.7653,Z 142,A -30.5472,B 23.1243,C -1.1926,E1 23.2952,E2 477.3219} C_DIS
LIN {X 111.9399,Y -55.4292,Z 142,A -28.9812,B 23.1244,C -1.1903,E1 23.2971,E2 475.7707} C_DIS
LIN {X 113.915,Y -51.2481,Z 142,A -26.8535,B 23.1241,C -1.197,E1 23.2996,E2 473.6385} C_DIS
LIN {X 115.2833,Y -48.0904,Z 142,A -25.2442,B 23.1238,C -1.2033,E1 23.3014,E2 472.0229} C_DIS
LIN {X 116.958,Y -43.8609,Z 142,A -23.2344,B 23.1236,C -1.2061,E1 23.3034,E2 470.0183} C_DIS
LIN {X 117.9241,Y -41.194,Z 142,A -21.8243,B 23.1232,C -1.2154,E1 23.3047,E2 468.5933} C_DIS
LIN {X 119.3031,Y -37.013,Z 142,A -20.09,B 23.1235,C -1.2079,E1 23.3062,E2 466.8885} C_DIS
LIN {X 120.2383,Y -33.8491,Z 142,A -18.3461,B 23.1227,C -1.2238,E1 23.3076,E2 465.1152} C_DIS
LIN {X 121.118,Y -30.5521,Z 142,A -15.7372,B 23.1199,C -1.2798,E1 23.3094,E2 462.381} C_DIS
LIN {X 122.6975,Y -23.416,Z 142,A -13.5405,B 23.1222,C -1.234,E1 23.3105,E2 460.3143} C_DIS
LIN {X 123.3613,Y -19.628,Z 142,A -11.7946,B 23.122,C -1.2388,E1 23.3113,E2 458.5674} C_DIS
LIN {X 123.854,Y -16.2234,Z 142,A -10.2276,B 23.1218,C -1.2434,E1 23.3119,E2 456.9989} C_DIS
LIN {X 124.2781,Y -12.5859,Z 142,A -8.4915,B 23.1213,C -1.2515,E1 23.3125,E2 455.2534} C_DIS
LIN {X 124.5857,Y -9.0243,Z 142,A -6.9216,B 23.1213,C -1.2535,E1 23.3128,E2 453.6887} C_DIS
LIN {X 124.8076,Y -5.1167,Z 142,A -5.0271,B 23.1207,C -1.2641,E1 23.313,E2 451.7796} C_DIS
LIN {X 124.9097,Y -0.9148,Z 142,A -3.25,B 23.1207,C -1.263,E1 23.3131,E2 450.0168} C_DIS
LIN {X 124.8856,Y 2.6352,Z 142,A -1.6065,B 23.1204,C -1.269,E1 23.3131,E2 448.3688} C_DIS
LIN {X 124.7143,Y 7.0549,Z 142,A 0.4826,B 23.12,C -1.2784,E1 23.3128,E2 446.2694} C_DIS
LIN {X 124.4511,Y 10.7238,Z 142,A 2.0534,B 23.12,C -1.2782,E1 23.3124,E2 444.7093} C_DIS
LIN {X 124.0564,Y 14.5972,Z 142,A 3.8451,B 23.1197,C -1.2842,E1 23.3119,E2 442.914} C_DIS
LIN {X 123.5702,Y 18.2697,Z 142,A 5.6064,B 23.1192,C -1.2926,E1 23.3112,E2 441.1428} C_DIS
LIN {X 122.9685,Y 21.9488,Z 142,A 7.2535,B 23.1191,C -1.2949,E1 23.3104,E2 439.5003} C_DIS
LIN {X 122.2031,Y 25.8771,Z 142,A 9.0996,B 23.1188,C -1.3012,E1 23.3094,E2 437.6501} C_DIS
LIN {X 121.3753,Y 29.5141,Z 142,A 10.7872,B 23.1185,C -1.3053,E1 23.3083,E2 435.9625} C_DIS
LIN {X 120.6719,Y 32.2687,Z 142,A 12.2755,B 23.1178,C -1.3182,E1 23.3072,E2 434.451} C_DIS
LIN {X 119.354,Y 36.8465,Z 142,A 14.2303,B 23.1181,C -1.3138,E1 23.3057,E2 432.5196} C_DIS
LIN {X 118.0769,Y 40.7533,Z 142,A 16.0629,B 23.1179,C -1.3169,E1 23.3041,E2 430.6904} C_DIS
LIN {X 116.9865,Y 43.7846,Z 142,A 17.6034,B 23.1175,C -1.3243,E1 23.3026,E2 429.1406} C_DIS
LIN {X 115.8547,Y 46.697,Z 142,A 19.1154,B 23.1171,C -1.3323,E1 23.301,E2 427.6175} C_DIS
LIN {X 114.1177,Y 50.795,Z 142,A 21.0413,B 23.1171,C -1.3326,E1 23.2989,E2 425.7023} C_DIS
LIN {X 112.614,Y 54.0468,Z 142,A 22.631,B 23.117,C -1.3347,E1 23.297,E2 424.1165} C_DIS
LIN {X 110.4976,Y 58.2514,Z 142,A 24.7776,B 23.1167,C -1.3401,E1 23.2942,E2 421.9687} C_DIS
LIN {X 108.6478,Y 61.6372,Z 142,A 26.4262,B 23.1167,C -1.3392,E1 23.292,E2 420.3318} C_DIS
LIN {X 106.232,Y 65.7135,Z 142,A 28.8199,B 23.1158,C -1.3554,E1 23.2885,E2 417.9103} C_DIS
LIN {X 103.7327,Y 69.5916,Z 142,A 30.8775,B 23.1157,C -1.3581,E1 23.2854,E2 415.8571} C_DIS
LIN {X 101.8583,Y 72.3079,Z 142,A 32.557,B 23.115,C -1.3698,E1 23.2827,E2 414.1569} C_DIS
LIN {X 98.9157,Y 76.2834,Z 142,A 34.3631,B 23.1159,C -1.3535,E1 23.2797,E2 412.4015} C_DIS
LIN {X 95.6818,Y 80.3018,Z 142,A 36.9903,B 23.1149,C -1.3714,E1 23.275,E2 409.7421} C_DIS
LIN {X 92.806,Y 83.6096,Z 142,A 39.0355,B 23.1146,C -1.3777,E1 23.2712,E2 407.6911} C_DIS
LIN {X 89.8527,Y 86.775,Z 142,A 40.9742,B 23.1144,C -1.3799,E1 23.2675,E2 405.756} C_DIS
LIN {X 86.6787,Y 89.946,Z 142,A 43.0266,B 23.1142,C -1.384,E1 23.2634,E2 403.7026} C_DIS
LIN {X 83.5776,Y 92.8347,Z 142,A 44.9965,B 23.1139,C -1.3892,E1 23.2593,E2 401.7282} C_DIS
LIN {X 80.1853,Y 95.7795,Z 142,A 46.9953,B 23.1139,C -1.3903,E1 23.2551,E2 399.735} C_DIS
LIN {X 77.1234,Y 98.2618,Z 142,A 49.0002,B 23.1131,C -1.4029,E1 23.2507,E2 397.7064} C_DIS
LIN {X 72.955,Y 101.3957,Z 142,A 50.9109,B 23.1142,C -1.3847,E1 23.2465,E2 395.8492} C_DIS
LIN {X 67.7647,Y 104.9353,Z 142,A 54.0002,B 23.1134,C -1.399,E1 23.2393,E2 392.7349} C_DIS
LIN {X 64.2646,Y 107.1148,Z 142,A 55.9845,B 23.1129,C -1.4062,E1 23.2345,E2 390.7392} C_DIS
LIN {X 59.3669,Y 109.9047,Z 142,A 58.5454,B 23.1128,C -1.4087,E1 23.2283,E2 388.1801} C_DIS
LIN {X 56.4827,Y 111.4121,Z 142,A 60.1248,B 23.1125,C -1.4147,E1 23.2243,E2 386.5902} C_DIS
LIN {X 52.593,Y 113.3002,Z 142,A 61.9126,B 23.1128,C -1.4081,E1 23.2199,E2 384.8242} C_DIS
LIN {X 49.5524,Y 114.6625,Z 142,A 63.4488,B 23.1128,C -1.4102,E1 23.2159,E2 383.2867} C_DIS
LIN {X 46.141,Y 116.0789,Z 142,A 65.3959,B 23.1119,C -1.4235,E1 23.2108,E2 381.3106} C_DIS
LIN {X 41.349,Y 117.8703,Z 142,A 67.4385,B 23.1126,C -1.4118,E1 23.2056,E2 379.3024} C_DIS
LIN {X 38.387,Y 118.8678,Z 142,A 68.8514,B 23.1126,C -1.4121,E1 23.2018,E2 377.8918} C_DIS
LIN {X 35.1201,Y 119.873,Z 142,A 70.3882,B 23.1126,C -1.4119,E1 23.1977,E2 376.3584} C_DIS
LIN {X 31.235,Y 120.9447,Z 142,A 72.3653,B 23.1122,C -1.4189,E1 23.1923,E2 374.3669} C_DIS
LIN {X 28.2766,Y 121.6701,Z 142,A 73.8649,B 23.1119,C -1.4243,E1 23.1882,E2 372.8558} C_DIS
LIN {X 23.7097,Y 122.6414,Z 142,A 75.8911,B 23.1121,C -1.4201,E1 23.1827,E2 370.843} C_DIS
LIN {X 19.7013,Y 123.35,Z 142,A 77.7749,B 23.1121,C -1.4215,E1 23.1775,E2 368.9578} C_DIS
LIN {X 16.2106,Y 123.8557,Z 142,A 79.3304,B 23.1121,C -1.4192,E1 23.1732,E2 367.4097} C_DIS
LIN {X 12.2407,Y 124.3112,Z 142,A 81.2007,B 23.1121,C -1.4211,E1 23.168,E2 365.5358} C_DIS
LIN {X 8.4624,Y 124.6267,Z 142,A 82.9633,B 23.1121,C -1.4223,E1 23.1631,E2 363.7712} C_DIS
LIN {X 4.8304,Y 124.8187,Z 142,A 84.5646,B 23.1121,C -1.4193,E1 23.1587,E2 362.1781} C_DIS
LIN {X 1.0374,Y 124.9084,Z 142,A 86.3351,B 23.1121,C -1.4204,E1 23.1537,E2 360.4051} C_DIS
LIN {X -2.5672,Y 124.8868,Z 142,A 88.0455,B 23.112,C -1.4225,E1 23.1489,E2 358.6891} C_DIS
LIN {X -6.1266,Y 124.7619,Z 142,A 89.5999,B 23.1122,C -1.4185,E1 23.1446,E2 357.1446} C_DIS
LIN {X -10.0106,Y 124.5113,Z 142,A 91.4252,B 23.1122,C -1.4196,E1 23.1395,E2 355.3159} C_DIS
LIN {X -13.5886,Y 124.1709,Z 142,A 93.0222,B 23.1124,C -1.4165,E1 23.1351,E2 353.7258} C_DIS
LIN {X -17.2807,Y 123.7115,Z 142,A 94.7857,B 23.1123,C -1.4179,E1 23.1302,E2 351.9571} C_DIS
LIN {X -20.8206,Y 123.1648,Z 142,A 96.466,B 23.1123,C -1.4184,E1 23.1256,E2 350.2738} C_DIS
LIN {X -24.9373,Y 122.3974,Z 142,A 98.3227,B 23.1125,C -1.4141,E1 23.1205,E2 348.4259} C_DIS
LIN {X -27.954,Y 121.7439,Z 142,A 100.3472,B 23.111,C -1.4394,E1 23.1148,E2 346.3339} C_DIS
LIN {X -32.5367,Y 120.6004,Z 142,A 101.9646,B 23.1125,C -1.4133,E1 23.1106,E2 344.7805} C_DIS
LIN {X -36.2753,Y 119.5288,Z 142,A 103.4571,B 23.1134,C -1.3988,E1 23.1067,E2 343.3223} C_DIS
LIN {X -41.6967,Y 117.749,Z 142,A 106.4453,B 23.1126,C -1.4116,E1 23.0987,E2 340.2955} C_DIS
LIN {X -46.1593,Y 116.0715,Z 142,A 108.4897,B 23.1132,C -1.4026,E1 23.0934,E2 338.2693} C_DIS
LIN {X -49.3532,Y 114.7486,Z 142,A 110.0948,B 23.1132,C -1.4012,E1 23.0893,E2 336.6637} C_DIS
LIN {X -52.2799,Y 113.445,Z 142,A 111.557,B 23.1134,C -1.3987,E1 23.0856,E2 335.2041} C_DIS
LIN {X -57.4826,Y 110.9013,Z 142,A 114.1615,B 23.1137,C -1.3922,E1 23.0791,E2 332.6087} C_DIS
LIN {X -63.2793,Y 107.6992,Z 142,A 117.6645,B 23.1129,C -1.4067,E1 23.0705,E2 329.0574} C_DIS
LIN {X -66.325,Y 105.8515,Z 142,A 119.0491,B 23.1137,C -1.393,E1 23.0673,E2 327.703} C_DIS
LIN {X -70.0597,Y 103.4168,Z 142,A 121.0582,B 23.114,C -1.3876,E1 23.0626,E2 325.7007} C_DIS
LIN {X -73.6656,Y 100.8806,Z 142,A 123.1419,B 23.114,C -1.3861,E1 23.0579,E2 323.6129} C_DIS
LIN {X -77.3038,Y 98.12,Z 142,A 125.179,B 23.1145,C -1.3792,E1 23.0534,E2 321.5852} C_DIS
LIN {X -80.522,Y 95.4971,Z 142,A 126.8417,B 23.1153,C -1.3649,E1 23.0499,E2 319.9522} C_DIS
LIN {X -83.0386,Y 93.3173,Z 142,A 128.6619,B 23.1148,C -1.3737,E1 23.046,E2 318.1017} C_DIS
LIN {X -86.1065,Y 90.4938,Z 142,A 130.5711,B 23.115,C -1.3691,E1 23.0421,E2 316.1957} C_DIS
LIN {X -89.0251,Y 87.624,Z 142,A 132.3076,B 23.1156,C -1.3587,E1 23.0387,E2 314.4778} C_DIS
LIN {X -91.0431,Y 85.5255,Z 142,A 133.8401,B 23.1154,C -1.3637,E1 23.0357,E2 312.9254} C_DIS
LIN {X -93.9701,Y 82.2985,Z 142,A 135.8155,B 23.1157,C -1.3576,E1 23.0321,E2 310.9557} C_DIS
LIN {X -96.6774,Y 79.1004,Z 142,A 137.739,B 23.116,C -1.3527,E1 23.0286,E2 309.0352} C_DIS
LIN {X -99.4304,Y 75.6116,Z 142,A 139.8404,B 23.1161,C -1.3499,E1 23.025,E2 306.93} C_DIS
LIN {X -102.0626,Y 72.0182,Z 142,A 141.8587,B 23.1165,C -1.3433,E1 23.0218,E2 304.9179} C_DIS
LIN {X -104.5594,Y 68.3438,Z 142,A 143.9583,B 23.1166,C -1.3402,E1 23.0185,E2 302.8148} C_DIS
LIN {X -106.8934,Y 64.6312,Z 142,A 145.9397,B 23.117,C -1.3333,E1 23.0156,E2 300.8401} C_DIS
LIN {X -110.1367,Y 58.9352,Z 142,A 149.0118,B 23.1174,C -1.3272,E1 23.0114,E2 297.7659} C_DIS
LIN {X -111.9307,Y 55.4479,Z 142,A 150.6924,B 23.1179,C -1.317,E1 23.0093,E2 296.1015} C_DIS
LIN {X -113.3814,Y 52.4173,Z 142,A 152.658,B 23.1172,C -1.33,E1 23.007,E2 294.0911} C_DIS
LIN {X -114.9534,Y 48.8796,Z 142,A 154.0612,B 23.1183,C -1.3092,E1 23.0055,E2 292.7328} C_DIS
LIN {X -116.4253,Y 45.2559,Z 142,A 155.8135,B 23.1187,C -1.302,E1 23.0037,E2 290.9883} C_DIS
LIN {X -117.5438,Y 42.2658,Z 142,A 157.2965,B 23.1189,C -1.2982,E1 23.0023,E2 289.5058} C_DIS
LIN {X -118.6465,Y 39.0656,Z 142,A 158.8904,B 23.1191,C -1.2951,E1 23.0008,E2 287.91} C_DIS
LIN {X -119.8373,Y 35.2419,Z 142,A 160.7191,B 23.1194,C -1.289,E1 22.9994,E2 286.0854} C_DIS
LIN {X -120.8951,Y 31.4306,Z 142,A 162.711,B 23.1194,C -1.2905,E1 22.9979,E2 284.0769} C_DIS
LIN {X -121.9286,Y 27.1443,Z 142,A 164.7107,B 23.1197,C -1.2832,E1 22.9966,E2 282.0833} C_DIS
LIN {X -122.7691,Y 23.0414,Z 142,A 166.6319,B 23.12,C -1.277,E1 22.9956,E2 280.1654} C_DIS
LIN {X -123.4599,Y 18.9916,Z 142,A 168.9242,B 23.1195,C -1.2879,E1 22.9946,E2 277.8304} C_DIS
LIN {X -124.02,Y 14.9019,Z 142,A 170.7188,B 23.12,C -1.2777,E1 22.994,E2 276.0502} C_DIS
LIN {X -124.41,Y 11.2104,Z 142,A 172.1661,B 23.1208,C -1.2616,E1 22.9936,E2 274.6348} C_DIS
LIN {X -124.6964,Y 7.3454,Z 142,A 173.9222,B 23.1212,C -1.255,E1 22.9933,E2 272.884} C_DIS
LIN {X -124.867,Y 3.3628,Z 142,A 175.7253,B 23.1215,C -1.248,E1 22.9932,E2 271.0868} C_DIS
LIN {X -124.9122,Y -0.4954,Z 142,A 177.5301,B 23.1217,C -1.2438,E1 22.9932,E2 269.2811} C_DIS
LIN {X -124.8251,Y -4.6669,Z 142,A 179.4154,B 23.1221,C -1.2364,E1 22.9932,E2 267.4022} C_DIS
LIN {X -124.6042,Y -8.7708,Z 142,A -178.6651,B 23.1224,C -1.2318,E1 22.9936,E2 265.4819} C_DIS
LIN {X -124.2847,Y -12.5176,Z 142,A -176.9278,B 23.1226,C -1.2268,E1 22.9941,E2 263.7461} C_DIS
LIN {X -123.8535,Y -16.2273,Z 142,A -175.2457,B 23.1229,C -1.2201,E1 22.9946,E2 262.0702} C_DIS
LIN {X -123.3698,Y -19.5732,Z 142,A -173.1896,B 23.1221,C -1.2362,E1 22.9956,E2 259.9595} C_DIS
LIN {X -122.67,Y -23.5598,Z 142,A -171.0758,B 23.1219,C -1.2412,E1 22.9967,E2 257.8193} C_DIS
LIN {X -121.5558,Y -28.765,Z 142,A -169.2848,B 23.1236,C -1.2064,E1 22.9978,E2 256.1059} C_DIS
LIN {X -120.729,Y -32.0545,Z 142,A -167.8557,B 23.1241,C -1.1964,E1 22.9988,E2 254.6933} C_DIS
LIN {X -119.9848,Y -34.7383,Z 142,A -166.0966,B 23.1233,C -1.2126,E1 23.0002,E2 252.8818} C_DIS
LIN {X -118.9207,Y -38.2213,Z 142,A -164.809,B 23.1243,C -1.1916,E1 23.0012,E2 251.64} C_DIS
LIN {X -117.6835,Y -41.8784,Z 142,A -162.9723,B 23.1245,C -1.189,E1 23.0029,E2 249.7984} C_DIS
LIN {X -116.4587,Y -45.1698,Z 142,A -161.4588,B 23.1249,C -1.1802,E1 23.0044,E2 248.298} C_DIS
LIN {X -115.2937,Y -48.0655,Z 142,A -160.0429,B 23.1251,C -1.1754,E1 23.0059,E2 246.886} C_DIS
LIN {X -114.2378,Y -50.5265,Z 142,A -158.5815,B 23.1248,C -1.1816,E1 23.0076,E2 245.3999} C_DIS
LIN {X -111.389,Y -56.5281,Z 142,A -155.6566,B 23.1255,C -1.1679,E1 23.0111,E2 242.4927} C_DIS
LIN {X -109.7642,Y -59.626,Z 142,A -154.0444,B 23.1257,C -1.1638,E1 23.0132,E2 240.8819} C_DIS
LIN {X -107.8715,Y -62.986,Z 142,A -152.1546,B 23.1257,C -1.1641,E1 23.0159,E2 238.9805} C_DIS
LIN {X -105.515,Y -66.8582,Z 142,A -150.2808,B 23.1263,C -1.15,E1 23.0186,E2 237.1323} C_DIS
LIN {X -103.4074,Y -70.0736,Z 142,A -148.3315,B 23.1262,C -1.1533,E1 23.0216,E2 235.164} C_DIS
LIN {X -100.9608,Y -73.5554,Z 142,A -146.3483,B 23.1263,C -1.1497,E1 23.0249,E2 233.1794} C_DIS
LIN {X -98.1615,Y -77.251,Z 142,A -144.1687,B 23.1265,C -1.1468,E1 23.0286,E2 230.9959} C_DIS
LIN {X -95.3184,Y -80.7332,Z 142,A -142.1519,B 23.1268,C -1.14,E1 23.0322,E2 228.9863} C_DIS
LIN {X -92.541,Y -83.902,Z 142,A -140.2048,B 23.127,C -1.1363,E1 23.0358,E2 227.0393} C_DIS
LIN {X -89.5122,Y -87.1268,Z 142,A -138.1744,B 23.1272,C -1.1319,E1 23.0397,E2 225.0106} C_DIS
LIN {X -86.5867,Y -90.0349,Z 142,A -136.2188,B 23.1272,C -1.1306,E1 23.0436,E2 223.0493} C_DIS
LIN {X -83.2833,Y -93.0983,Z 142,A -134.1978,B 23.1275,C -1.1245,E1 23.0478,E2 221.035} C_DIS
Enddeposition()
END
